(* Stoppen von Stationsfunktionen von rechter Arbeitsstation *)
	IF xStationStopWorkRight THEN
		(* Step  function station stop  *)
		CASE iStepAction OF
		(* Überprüfe zuerst welche Stationen gestoppt werden müssen  *)
		1:	iCheckStationNr:=1;
			ptrActivStation_FunctionStop:=ADR(TStation_Work_St1);
			iStepAction:=10;
		10:	IF (iCheckStationNr = 1) THEN ptrActivStation_FunctionStop:=ADR(TStation_Work_St1);
			ELSE
				iStepAction:=30;
				iCheckStationNr:=1;
				iStationNrReady:=0;
				RETURN;
			END_IF;
			xTmp:=	NOT(ptrActivStation_FunctionStop^.TControl.xDone)
					AND ptrActivStation_FunctionStop^.TControl.xRdy
					AND NOT(ptrActivStation_FunctionStop^.TControl.xExecute)
					AND NOT(ptrActivStation_FunctionStop^.TControl.xError)
					AND NOT(ptrActivStation_FunctionStop^.TControl.xStop);
			IF xTmp THEN
				(* Mindestens eine Station kann gestoppt werden *)
				iStepAction:=20;
			ELSE
				iCheckStationNr:=iCheckStationNr + 1;
			END_IF
		20:	ptrActivStation_FunctionStop^.TControl.xStop:=TRUE;
			iCheckStationNr:=iCheckStationNr + 1;
			(* next step *)
			iStepAction:=10;
		30:	IF (iCheckStationNr = 1) THEN ptrActivStation_FunctionStop:=ADR(TStation_Work_St1);END_IF;
			xTmp:=	(ptrActivStation_FunctionStop^.TControl.xDone OR ptrActivStation_FunctionStop^.TControl.xError)
					AND ptrActivStation_FunctionStop^.TControl.xRdy
					AND NOT(ptrActivStation_FunctionStop^.TControl.xExecute);
			IF xTmp THEN
				iStationNrReady:=iStationNrReady + 1;
			END_IF;
			iCheckStationNr:=iCheckStationNr + 1;
			IF (iCheckStationNr > 7) THEN
				IF (iStationNrReady = 7) THEN
					(* Alle Stationen sind gestoppt *)
					(* next step *)
					iStepAction:=40;
				ELSE
					(* Mindestens eine Station ist noch nicht gestoppt *)
					iCheckStationNr:=1;
					iStationNrReady:=0;
				END_IF;
			END_IF;
		(* Alle Stationen sind gestoppt. Nun müssen noch alle Achsen überprüft werden ob sie gestoppt sind *)
		40:	IF NOT(ptrTAxisZ_St1^.T_CtrleSingle.xNotMoving) AND NOT(ptrTAxisZ_St1^.T_CtrleSingle.xErr) THEN
				ptrTAxisZ_St1^.T_CtrleSingle.iFunction:=5;
				ptrTAxisZ_St1^.T_CtrleSingle.xExecute:=TRUE;
			END_IF;
			IF NOT(ptrTAxisS_St1^.T_CtrleSingle.xNotMoving) AND NOT(ptrTAxisS_St1^.T_CtrleSingle.xErr) THEN
				ptrTAxisS_St1^.T_CtrleSingle.iFunction:=5;
				ptrTAxisS_St1^.T_CtrleSingle.xExecute:=TRUE;
			END_IF;
			iStepAction:=50;
		(* Warte bis alle Achsen stehen *)
		50:	xTmp:=	(NOT(ptrTAxisZ_St1^.T_CtrleSingle.xExecute) AND (ptrTAxisZ_St1^.T_CtrleSingle.xDone OR ptrTAxisZ_St1^.T_CtrleSingle.xErr)) AND
					(NOT(ptrTAxisS_St1^.T_CtrleSingle.xExecute) AND (ptrTAxisS_St1^.T_CtrleSingle.xDone OR ptrTAxisS_St1^.T_CtrleSingle.xErr));
			IF xTmp THEN
				(* action done *)
				iStepAction:=90;
				T_ExchgParam.T_Visu.T_Message.iState:=274;	(* Warnung: Funktion wurde gestoppt ! *)
			END_IF;
		(* action done *)
		90:	T_Visu.T_CtrleAction.xFunctionActive:=FALSE;
			T_StartUp.T_State.xBlockChangeMovementVisu:=FALSE;
			T_Visu.T_CtrleAction.xDone:=TRUE;
			T_Visu.T_CtrleAction.xNotReady:=FALSE;
			T_Visu.T_CtrleAction.xErr:=FALSE;
			T_Visu.T_CtrleAction.udiErrorID:=0;
			xStationStopWorkRight:=FALSE;
		(* function not ready *)
		95:	T_StartUp.T_State.xBlockChangeMovementVisu:=FALSE;
			TimerNotReady(IN:=TRUE);
			xStationStopWorkRight:=FALSE;
		END_CASE;
	END_IF;
END_ACTION
ACTION VisuFunction_ToolCalibration:
(* Ausführen der Stationsfunktion für das Kalibrieren des ToolDefelction und ToolTorque *)
	IF xStationToolCalibrateFunction THEN
		(* Step  function station  *)
		CASE iStepAction OF
		(* Überprüfe zuerst ob es sich um die Station MicroHead oder Entgratstation handelt  *)
		1:	IF (T_ExchgParam.T_StationCommon.T_Param_StationWork.T_Fct_SpindleCalibration.iSelectCalibrationCylinder = 1) THEN
				ptrActivStation^.THWWorkStation.TCtrlWork.xActiveCalibrateToolDeflection:=TRUE;
				ptrActivStation^.THWWorkStation.TCtrlWork.xActiveCalibrateToolTorque:=FALSE;
			END_IF;
			IF (T_ExchgParam.T_StationCommon.T_Param_StationWork.T_Fct_SpindleCalibration.iSelectCalibrationCylinder = 2) THEN
				ptrActivStation^.THWWorkStation.TCtrlWork.xActiveCalibrateToolDeflection:=FALSE;
				ptrActivStation^.THWWorkStation.TCtrlWork.xActiveCalibrateToolTorque:=TRUE;
			END_IF;
			iStepAction:=10;
		(* check station state *)
		10:	xTmp:=	ptrActivStation^.TControl.xDone
					AND ptrActivStation^.TControl.xRdy
					AND NOT(ptrActivStation^.TControl.xExecute)
					AND NOT(ptrActivStation^.TControl.xError)
					AND NOT(ptrActivStation^.TControl.xStop);
			(* next step *)
			IF xTmp THEN iStepAction:=20; ELSE iStepAction:=95; END_IF
		(* determin function number *)
		20:	T_ExchgParam.T_Visu.T_Message.iState:=66;	(* Info: Kalibrierungsfunktion gestartet ! *)
			ptrActivStation^.TControl.iFunctNr:=7;
			ptrActivStation^.TControl.xExecute:=TRUE;
			ptrActivStation^.THWWorkStation.TCtrlWork.xStopToolRotation:=TRUE;
			iStepAction:=30;
			(* next step *)
			xStepActionDone:=FALSE;
		(* wait confirmation *)
		30:	IF NOT(xStepActionDone) THEN
			(* release execution *)
				ptrActivStation^.TControl.xExecute:=FALSE;
				xStepActionDone:=TRUE;
			ELSE
				T_ExchgParam.T_StationCommon.T_Param_StationWork.T_Fct_SpindleCalibration:=T_NovRAM.T_Parameter.T_StationWork[gciStationSt1].T_Fct_SpindleCalibration;
				IF (T_ExchgParam.T_StationCommon.T_Param_StationWork.T_Fct_SpindleCalibration.iSelectCalibrationCylinder = 1) THEN
					T_ExchgParam.T_StationCommon.T_Param_StationWork.T_Fct_SpindleCalibration.arOffsetToolDeflection[1]:=ptrActivStation^.THWWorkStation.TCtrlWork.rOffsetToolDeflection;
				END_IF;
				IF (T_ExchgParam.T_StationCommon.T_Param_StationWork.T_Fct_SpindleCalibration.iSelectCalibrationCylinder = 2) THEN
					T_ExchgParam.T_StationCommon.T_Param_StationWork.T_Fct_SpindleCalibration.arOffseTToolTorque[1]:=ptrActivStation^.THWWorkStation.TCtrlWork.rOffseTToolTorque;
				END_IF;
				IF ptrActivStation^.TControl.xDone THEN
					(* action done *)
					iStepAction:=40;
					xStepActionDone:=FALSE;
				END_IF
			END_IF
		40:	T_ExchgParam.T_StationCommon.T_Param_StationWork.T_Fct_SpindleCalibration:=T_NovRAM.T_Parameter.T_StationWork[gciStationSt1].T_Fct_SpindleCalibration;
			iStepAction:=50;
		50:	xAction_SaveNovRAM:=TRUE;
			xBlockSetNovRamAction_End:=TRUE;
			iStepActionNovRam:=1;
			iStepAction:=60;
		60:	IF NOT(xAction_SaveNovRAM) THEN
				T_ExchgParam.T_Visu.T_Message.iState:=67;	(* Info: Kalibrierungsfunktion beendet ! *)
				xUpdateStationParameter:=TRUE;
				iStepAction:=90;
			END_IF;
		(* action done *)
		90:	T_Visu.T_CtrleAction.xDone:=TRUE;
			T_Visu.T_CtrleAction.xNotReady:=FALSE;
			T_Visu.T_CtrleAction.xErr:=FALSE;
			T_Visu.T_CtrleAction.udiErrorID:=0;
			xStationToolCalibrateFunction:=FALSE;
		(* function not ready *)
		95:	TimerNotReady(IN:=TRUE);
			xStationToolCalibrateFunction:=FALSE;
		END_CASE
	END_IF

(* Spindelkalibrierung EIN/AUS *)
	IF xSpindelCalibrationONOFF THEN
		CASE iStepAction OF
		(* check state *)
		1:	xTmp:=	TRUE;
			(* next step *)
			IF xTmp THEN iStepAction:=10; ELSE iStepAction:=95; END_IF
		(* Set Value *)
		10:	gxSpindelCalibrationONOFF_St1:=NOT(gxSpindelCalibrationONOFF_St1);
			iStepAction:=90;
		(* action done *)
		90:	T_Visu.T_CtrleAction.xDone:=TRUE;
			T_Visu.T_CtrleAction.xNotReady:=FALSE;
			T_Visu.T_CtrleAction.xErr:=FALSE;
			T_Visu.T_CtrleAction.udiErrorID:=0;
			xSpindelCalibrationONOFF:=FALSE;
		(* cylinder not ready *)
		95:	TimerNotReady(IN:=TRUE);
			xSpindelCalibrationONOFF:=FALSE;
		END_CASE
	END_IF;

	IF (T_Visu.T_PlcParam.dwActualPage = gT_PageNumber.iWorkStation_Setup1) THEN
		IF (T_NovRAM.T_Parameter.T_StationWork[gciStationSt1].T_Fct_SpindleCalibration.iSelectCalibrationCylinder <> 1) AND
			(T_NovRAM.T_Parameter.T_StationWork[gciStationSt1].T_Fct_SpindleCalibration.iSelectCalibrationCylinder <> 2) THEN
			T_NovRAM.T_Parameter.T_StationWork[gciStationSt1].T_Fct_SpindleCalibration.iSelectCalibrationCylinder:=1;
		END_IF;
		IF (T_ExchgParam.T_StationCommon.T_Param_StationWork.T_Fct_SpindleCalibration.iSelectCalibrationCylinder <> 1) AND
			(T_ExchgParam.T_StationCommon.T_Param_StationWork.T_Fct_SpindleCalibration.iSelectCalibrationCylinder <> 2) THEN
			T_ExchgParam.T_StationCommon.T_Param_StationWork.T_Fct_SpindleCalibration.iSelectCalibrationCylinder:=1;
		END_IF;
		IF (T_ExchgParam.T_StationCommon.T_Param_StationWork.T_Fct_SpindleCalibration.iSelectCalibrationCylinder <>
		     T_NovRAM.T_Parameter.T_StationWork[gciStationSt1].T_Fct_SpindleCalibration.iSelectCalibrationCylinder) THEN
			T_NovRAM.T_Parameter.T_StationWork[gciStationSt1].T_Fct_SpindleCalibration.iSelectCalibrationCylinder:=
											T_ExchgParam.T_StationCommon.T_Param_StationWork.T_Fct_SpindleCalibration.iSelectCalibrationCylinder;
		END_IF;

		T_ExchgParam.T_StationCommon.T_Param_StationWork.T_Fct_SpindleCalibration.rEffectiveForceToolDeflection:=
					T_NovRAM.T_Parameter.T_StationWork[gciStationSt1].T_OnlineChange.rForceDeflection +
					T_NovRAM.T_Parameter.T_StationWork[gciStationSt1].T_Fct_SpindleCalibration.arOffsetToolDeflection[1];
		T_ExchgParam.T_StationCommon.T_Param_StationWork.T_Fct_SpindleCalibration.rNullValueToolDeflection:=
					T_NovRAM.T_Parameter.T_StationWork[gciStationSt1].T_OnlineChange.rForceDeflection;

		T_ExchgParam.T_StationCommon.T_Param_StationWork.T_Fct_SpindleCalibration.rEffectiveForceToolTorque:=
					T_NovRAM.T_Parameter.T_StationWork[gciStationSt1].T_OnlineChange.rTorqueLevelHC +
					T_NovRAM.T_Parameter.T_StationWork[gciStationSt1].T_Fct_SpindleCalibration.arOffseTToolTorque[1];
		T_ExchgParam.T_StationCommon.T_Param_StationWork.T_Fct_SpindleCalibration.rNullValueToolTorque:=
					T_NovRAM.T_Parameter.T_StationWork[gciStationSt1].T_OnlineChange.rTorqueLevelHC;

		IF NOT(xStationToolCalibrateFunction) THEN
			T_ExchgParam.T_StationCommon.T_Param_StationWork.T_Fct_SpindleCalibration.arOffsetToolDeflection:=
					T_NovRAM.T_Parameter.T_StationWork[gciStationSt1].T_Fct_SpindleCalibration.arOffsetToolDeflection;
			T_ExchgParam.T_StationCommon.T_Param_StationWork.T_Fct_SpindleCalibration.arOffseTToolTorque:=
					T_NovRAM.T_Parameter.T_StationWork[gciStationSt1].T_Fct_SpindleCalibration.arOffseTToolTorque;
		END_IF;
	END_IF;
END_ACTION
ACTION VisuFunction_ToolChange:
(* Resetten des Werkzeugwechsel für den Automatik für Station 1,2,3 und 4-->braucht mindestens den OperatorLevel oder für das setzen der berechneten Z EndPosition *)
	IF xProcessStation1ResetToolChange OR xZSaveEndPosCalc THEN
		CASE iStepAction OF
		(* Überprüfe zuerst ob mindestens der OperatorLevel gesetzt ist *)
		1:	IF (T_ExchgParam.T_Visu.T_Level.iActLevel < 1) THEN
				T_ExchgParam.T_Visu.T_Message.iState:=217;	(* Warnung: Mindestens OperatorLevel wird benötigt ! *)
				iStepAction:=90;
			ELSE
				iStepAction:=10;
			END_IF;
		10:	T_ExchgParam.T_Visu.T_Message.iState:=103;	(* Aufforderung: Speichern bestätigen <Enter>, abbrechen <Esc> ? *)
			iStepAction:=20;
		(* waiting for key <Enter> or <Esc> *)
		20:	IF RisingEdgeKeyPanel_Enter.Q THEN
				iStepAction:=30;
			ELSE
				IF RisingEdgeKeyPanel_Esc.Q THEN
					iStepAction:=90;
					T_ExchgParam.T_Visu.T_Message.iState:=202;	(* Warnung: Aktion abgebrochen ! *)
				END_IF
			END_IF
			(* An other message has been displayed *)
			IF (T_ExchgParam.T_Visu.T_Message.iState<>103) AND (T_ExchgParam.T_Visu.T_Message.iState<>202) THEN iStepAction:=90; END_IF
		30:	IF xProcessStation1ResetToolChange THEN
				T_NovRam.T_Parameter.T_StationWork[1].T_ToolCounter.diToolCycleCounter:=0;
				T_ExchgParam.T_StationCommon.T_ToolCounter_St1.diToolCycleCounter:=0;
				IF NOT(gxProcessCylindricalAreaActive) THEN
					garPositionEndProcCalc[1]:=T_NovRam.T_Parameter.T_StationWork[1].T_StProcess.rPositionEndProc;
					T_ExchgParam.T_StationCommon.rPositionEndProcCalc:=T_NovRam.T_Parameter.T_StationWork[1].T_StProcess.rPositionEndProc;
				ELSE
					garPositionEndProcCalc[1]:=T_NovRam.T_Parameter.T_StationWork[1].T_StProcess.rZPositionCylindricalArea;
					T_ExchgParam.T_StationCommon.rPositionEndProcCalc:=T_NovRam.T_Parameter.T_StationWork[1].T_StProcess.rZPositionCylindricalArea;
				END_IF;
				garCentringEndProcCalc[1]:=T_NovRam.T_Parameter.T_StationWork[1].T_StProcess.rCentringPosZ1Axis;
				T_ExchgParam.T_StationCommon.rCentringEndProcCalc:=T_NovRam.T_Parameter.T_StationWork[1].T_StProcess.rCentringPosZ1Axis;
			ELSE
				IF (T_ExchgParam.T_StationCommon.bSelectShowIncValue = 0) THEN
					garPositionEndProcCalc[1]:=T_ExchgParam.T_StationCommon.rPositionEndProcCalc;
				ELSE
					garCentringEndProcCalc[1]:=T_ExchgParam.T_StationCommon.rCentringEndProcCalc;
				END_IF;
			END_IF;
			iStepAction:=40;
		40:	IF xZSaveEndPosCalc THEN
				IF (T_ExchgParam.T_StationCommon.bSelectShowIncValue = 0) THEN
					IF (garPositionEndProcCalc[1] <> T_ExchgParam.T_StationCommon.rPositionEndProcCalc) THEN
						T_ExchgParam.T_StationCommon.rPositionEndProcCalc:=garPositionEndProcCalc[1];
					END_IF;
				ELSE
					IF (garCentringEndProcCalc[1] <> T_ExchgParam.T_StationCommon.rCentringEndProcCalc) THEN
						T_ExchgParam.T_StationCommon.rCentringEndProcCalc:=garCentringEndProcCalc[1];
					END_IF;
				END_IF;
			END_IF;
			xAction_SaveNovRAM:=TRUE;
			xBlockSetNovRamAction_End:=TRUE;
			iStepActionNovRam:=1;
			iStepAction:=50;
		50:	IF NOT(xAction_SaveNovRAM) THEN
				iStepAction:=90;
				IF xProcessStation1ResetToolChange THEN
					T_ExchgParam.T_Visu.T_Message.iState:=68;	(* Info: WzZähler für Station 1 wurde zurückgesetzt ! *)
				ELSE
					T_ExchgParam.T_Visu.T_Message.iState:=69;	(* Info: Position gespeichert ! *)
				END_IF;
			END_IF;
		(* axis not ready *)
		95:	TimerNotReady(IN:=TRUE);
			xProcessStation1ResetToolChange:=xZSaveEndPosCalc:=FALSE;
		(* slow/fast configuration done *)
		90:	T_Visu.T_CtrleAction.xDone:=TRUE;
			T_Visu.T_CtrleAction.xNotReady:=FALSE;
			T_Visu.T_CtrleAction.xErr:=FALSE;
			T_Visu.T_CtrleAction.udiErrorID:=0;
			xProcessStation1ResetToolChange:=xZSaveEndPosCalc:=FALSE;
		END_CASE
	END_IF;


(* Umschalten Z Ink Wert für Bearbeitung oder Zentrierung *)
	IF xSelectZInkWorkInfo OR xSelectZInkCentringInfo THEN
		CASE iStepAction OF
		(* Überprüfe zuerst ob mindestens der OperatorLevel gesetzt ist *)
		1:	iStepAction:=10;
		10:	IF xSelectZInkWorkInfo THEN
				T_ExchgParam.T_StationCommon.bSelectShowIncValue:=0;
			ELSE
				T_ExchgParam.T_StationCommon.bSelectShowIncValue:=1;
			END_IF;
			iStepAction:=90;
		(* axis not ready *)
		95:	TimerNotReady(IN:=TRUE);
			xSelectZInkWorkInfo:=xSelectZInkCentringInfo:=FALSE;
		(* slow/fast configuration done *)
		90:	T_Visu.T_CtrleAction.xDone:=TRUE;
			T_Visu.T_CtrleAction.xNotReady:=FALSE;
			T_Visu.T_CtrleAction.xErr:=FALSE;
			T_Visu.T_CtrleAction.udiErrorID:=0;
			xSelectZInkWorkInfo:=xSelectZInkCentringInfo:=FALSE;
		END_CASE
	END_IF;
END_ACTION
ACTION VisuUpdateParameter:
IF (T_Visu.T_PlcParam.dwActualPage = gT_PageNumber.iHandMode_OnlineChange) THEN
	xFctUpdateOnlineChangeValue(	ptrProfileOnlineChange:=ADR(T_Profile.T_Profile_MinMax),
									ptrProfileOnlineChangeLoad:=ADR(T_Profile.T_LoadProfileParameter.T_ProfileOnlineChange),
									ptrExchgParamStationCommon:=ADR(T_ExchgParam.T_ProfileCommon.T_OnlineChange),
									TOnlineChangeParameter:=T_NovRam.T_Parameter.T_StationWork[gciStationSt1].T_OnlineChange);
END_IF;
END_ACTION

(* POU PRG_LAYER5_VISU/FB_VISU/FBQVIS_INITPAGE, ST *)
FUNCTION_BLOCK FBQVIS_INITPAGE
VAR_INPUT
END_VAR
VAR_OUTPUT
END_VAR
VAR_IN_OUT
	T_Visu:ST_QVIS;
END_VAR
VAR
(* pointer *)
	ptrConfigPage: POINTER TO ST_CONFIGPAGE;
(* variable *)
	iIndexPage:INT;
	iPageNumber:INT;
(* variable Tmp *)
	i:INT;
END_VAR
(****************************************************************************************************************************************************)
(***********                    This Functionblock init all the defined page in QVis for the hole page management                            ************)
(****************************************************************************************************************************************************)
(* init. index array *)
FOR i:=0 TO 999 DO
	T_Visu.T_PageIndex[i].iIndexConfigPage:=0;
END_FOR

(* init. Number Page *)
iPageNumber:=0;
Page_000_Start;
Page_001_BIOS;
Page_002_BIOS;
Page_010_AutoMode_Process;
Page_011_AutoMode_ProcessValue1;
Page_012_AutoMode_ProcessValue2;	(* IGS *)
Page_013_AutoMode_PartQuality;
Page_020_AutoMode_Referencing;
Page_030_AutoMode_Profile;
Page_040_AutoMode_ToolChange;
Page_041_AutoMode_UserLevel;
Page_042_AutoMode_Language;
Page_050_AutoMode_WPCounter;
Page_051_AutoMode_LampTest;
Page_052_AutoMode_SafetyCheck;
Page_053_AutoMode_SysInfo;
Page_060_AutoMode_ErrorList;
Page_070_AutoMode_Parameter;
Page_110_HandMode_Process;
Page_111_HandMode_WorkParameter;		(* IGS *)
Page_112_HandMode_RegulatorPara;		(* IGS *)
Page_113_HandMode_OnlineChange;
Page_114_HandMode_ConfigPosition;
Page_120_HandMode_ProfileMngmt1;
Page_150_HandMode_Setup1;
Page_160_HandMode_ErrorList;
Page_170_HandMode_Parameter;
Page_210_WorkStation_Axis1;
Page_220_WorkStation_Cylinder1;
Page_230_WorkStation_Valve1;
Page_240_WorkStation_Function1;
Page_250_WorkStation_Setup1;
Page_251_WorkStation_Setup2;
Page_252_WorkStation_Setup3;
Page_253_WorkStation_Setup4;
Page_254_WorkStation_Setup5;
Page_260_WorkStation_ErrorList;
Page_270_WorkStation_Parameter;
END_FUNCTION_BLOCK
ACTION Page_000_Start:
(* QVis page 0, start page *)
iIndexPage:=gT_PageNumber.iStart_Page1;
iPageNumber:=iPageNumber+1;
T_Visu.T_PageIndex[iIndexPage].iIndexConfigPage:=iPageNumber;
ptrConfigPage:=ADR(T_Visu.T_ConfigPage[T_Visu.T_PageIndex[iIndexPage].iIndexConfigPage]);
ptrConfigPage^.sName:='Start page';
ptrConfigPage^.wMaskBtPanelLeft:=16#0;
ptrConfigPage^.wMaskBtPanelRight:=16#0;
ptrConfigPage^.wMaskFunctionPanel:=16#0;
(* Navigation panel restriction *)
ptrConfigPage^.wMaskTouchScreenNavPanel:=16#0;
(* Process mask *)
ptrConfigPage^.wMaskProcBtPanelLeft:=16#0;
ptrConfigPage^.wMaskProcBtPanelRight:=16#0;
ptrConfigPage^.wMaskProcFunctionPanel:=16#0;
(* Button edge action *)
ptrConfigPage^.aiRTrigActionPanelLeft[1]:=0;
ptrConfigPage^.aiRTrigActionPanelLeft[2]:=0;
ptrConfigPage^.aiRTrigActionPanelLeft[3]:=0;
ptrConfigPage^.aiRTrigActionPanelLeft[4]:=0;
ptrConfigPage^.aiRTrigActionPanelLeft[5]:=0;
ptrConfigPage^.aiRTrigActionPanelRight[1]:=0;
ptrConfigPage^.aiRTrigActionPanelRight[2]:=0;
ptrConfigPage^.aiRTrigActionPanelRight[3]:=0;
ptrConfigPage^.aiRTrigActionPanelRight[4]:=0;
ptrConfigPage^.aiRTrigActionPanelRight[5]:=0;
ptrConfigPage^.aiFTrigActionPanelRight[1]:=0;
ptrConfigPage^.aiFTrigActionPanelRight[2]:=0;
ptrConfigPage^.aiFTrigActionPanelRight[3]:=0;
ptrConfigPage^.aiFTrigActionPanelRight[4]:=0;
ptrConfigPage^.aiFTrigActionPanelRight[5]:=0;
ptrConfigPage^.aiRTrigActionFunctionPanel[1]:=0;
ptrConfigPage^.aiRTrigActionFunctionPanel[2]:=0;
ptrConfigPage^.aiRTrigActionFunctionPanel[3]:=0;
ptrConfigPage^.aiRTrigActionFunctionPanel[4]:=0;
ptrConfigPage^.aiRTrigActionFunctionPanel[5]:=0;
ptrConfigPage^.aiRTrigActionFunctionPanel[6]:=0;
ptrConfigPage^.aiRTrigActionFunctionPanel[7]:=0;
ptrConfigPage^.aiRTrigActionFunctionPanel[8]:=0;
ptrConfigPage^.aiRTrigActionFunctionPanel[9]:=0;
ptrConfigPage^.aiRTrigActionFunctionPanel[10]:=0;
ptrConfigPage^.aiRTrigActionFunctionPanel[11]:=0;
ptrConfigPage^.aiRTrigActionFunctionPanel[12]:=0;
ptrConfigPage^.aiRTrigActionTouchScreenNavPanel[1,1]:=0;
ptrConfigPage^.aiRTrigActionTouchScreenNavPanel[1,2]:=0;
ptrConfigPage^.aiRTrigActionTouchScreenNavPanel[1,3]:=0;
ptrConfigPage^.aiRTrigActionTouchScreenNavPanel[1,4]:=0;
ptrConfigPage^.aiRTrigActionTouchScreenNavPanel[1,5]:=0;
ptrConfigPage^.aiRTrigActionTouchScreenNavPanel[1,6]:=0;
ptrConfigPage^.aiRTrigActionTouchScreenNavPanel[1,7]:=0;
ptrConfigPage^.aiRTrigActionTouchScreenNavPanel[1,8]:=0;
ptrConfigPage^.aiRTrigActionTouchScreenNavPanel[1,9]:=0;
ptrConfigPage^.aiRTrigActionTouchScreenNavPanel[2,1]:=0;
ptrConfigPage^.aiRTrigActionTouchScreenNavPanel[2,2]:=0;
ptrConfigPage^.aiRTrigActionTouchScreenNavPanel[2,3]:=0;
ptrConfigPage^.aiRTrigActionTouchScreenNavPanel[2,4]:=0;
ptrConfigPage^.aiRTrigActionTouchScreenNavPanel[2,5]:=0;
ptrConfigPage^.aiRTrigActionTouchScreenNavPanel[2,6]:=0;
ptrConfigPage^.aiRTrigActionTouchScreenNavPanel[2,7]:=0;
ptrConfigPage^.aiRTrigActionTouchScreenNavPanel[2,8]:=0;
ptrConfigPage^.aiRTrigActionTouchScreenNavPanel[2,9]:=0;
ptrConfigPage^.aiRTrigActionTouchScreenNavPanel[3,1]:=0;
ptrConfigPage^.aiRTrigActionTouchScreenNavPanel[3,2]:=0;
ptrConfigPage^.aiRTrigActionTouchScreenNavPanel[3,3]:=0;
ptrConfigPage^.aiRTrigActionTouchScreenNavPanel[3,4]:=0;
ptrConfigPage^.aiRTrigActionTouchScreenNavPanel[3,5]:=0;
ptrConfigPage^.aiRTrigActionTouchScreenNavPanel[3,6]:=0;
ptrConfigPage^.aiRTrigActionTouchScreenNavPanel[3,7]:=0;
ptrConfigPage^.aiRTrigActionTouchScreenNavPanel[3,8]:=0;
ptrConfigPage^.aiRTrigActionTouchScreenNavPanel[3,9]:=0;
ptrConfigPage^.aiRTrigActionTouchScreenNavPanel[4,1]:=0;
ptrConfigPage^.aiRTrigActionTouchScreenNavPanel[4,2]:=0;
ptrConfigPage^.aiRTrigActionTouchScreenNavPanel[4,3]:=0;
ptrConfigPage^.aiRTrigActionTouchScreenNavPanel[4,4]:=0;
ptrConfigPage^.aiRTrigActionTouchScreenNavPanel[4,5]:=0;
ptrConfigPage^.aiRTrigActionTouchScreenNavPanel[4,6]:=0;
ptrConfigPage^.aiRTrigActionTouchScreenNavPanel[4,7]:=0;
ptrConfigPage^.aiRTrigActionTouchScreenNavPanel[4,8]:=0;
ptrConfigPage^.aiRTrigActionTouchScreenNavPanel[4,9]:=0;
ptrConfigPage^.aiRTrigActionTouchScreenNavPanel[5,1]:=0;
ptrConfigPage^.aiRTrigActionTouchScreenNavPanel[5,2]:=0;
ptrConfigPage^.aiRTrigActionTouchScreenNavPanel[5,3]:=0;
ptrConfigPage^.aiRTrigActionTouchScreenNavPanel[5,4]:=0;
ptrConfigPage^.aiRTrigActionTouchScreenNavPanel[5,5]:=0;
ptrConfigPage^.aiRTrigActionTouchScreenNavPanel[5,6]:=0;
ptrConfigPage^.aiRTrigActionTouchScreenNavPanel[5,7]:=0;
ptrConfigPage^.aiRTrigActionTouchScreenNavPanel[5,8]:=0;
ptrConfigPage^.aiRTrigActionTouchScreenNavPanel[5,9]:=0;
ptrConfigPage^.aiRTrigActionTouchScreenNavPanel[6,1]:=0;
ptrConfigPage^.aiRTrigActionTouchScreenNavPanel[6,2]:=0;
ptrConfigPage^.aiRTrigActionTouchScreenNavPanel[6,3]:=0;
ptrConfigPage^.aiRTrigActionTouchScreenNavPanel[6,4]:=0;
ptrConfigPage^.aiRTrigActionTouchScreenNavPanel[6,5]:=0;
ptrConfigPage^.aiRTrigActionTouchScreenNavPanel[6,6]:=0;
ptrConfigPage^.aiRTrigActionTouchScreenNavPanel[6,7]:=0;
ptrConfigPage^.aiRTrigActionTouchScreenNavPanel[6,8]:=0;
ptrConfigPage^.aiRTrigActionTouchScreenNavPanel[6,9]:=0;
ptrConfigPage^.xMaskBtStart:=TRUE;
ptrConfigPage^.xMaskBtStop:=FALSE;
END_ACTION
ACTION Page_001_BIOS:
(* QVis page 1, BIOS input Password *)
iIndexPage:=gT_PageNumber.iBIOS_Page1;
iPageNumber:=iPageNumber+1;
T_Visu.T_PageIndex[iIndexPage].iIndexConfigPage:=iPageNumber;
ptrConfigPage:=ADR(T_Visu.T_ConfigPage[T_Visu.T_PageIndex[iIndexPage].iIndexConfigPage]);
ptrConfigPage^.sName:='BIOS input Password';
ptrConfigPage^.wMaskBtPanelLeft:=16#0;
ptrConfigPage^.wMaskBtPanelRight:=16#0;
ptrConfigPage^.wMaskFunctionPanel:=16#0;
(* Navigation panel restriction *)
ptrConfigPage^.wMaskTouchScreenNavPanel:=16#0;
(* Process mask *)
ptrConfigPage^.wMaskProcBtPanelLeft:=16#0;
ptrConfigPage^.wMaskProcBtPanelRight:=16#0;
ptrConfigPage^.wMaskProcFunctionPanel:=16#0;
(* Button edge action *)
ptrConfigPage^.aiRTrigActionPanelLeft[1]:=0;
ptrConfigPage^.aiRTrigActionPanelLeft[2]:=0;
ptrConfigPage^.aiRTrigActionPanelLeft[3]:=0;
ptrConfigPage^.aiRTrigActionPanelLeft[4]:=0;
ptrConfigPage^.aiRTrigActionPanelLeft[5]:=0;
ptrConfigPage^.aiRTrigActionPanelRight[1]:=0;
ptrConfigPage^.aiRTrigActionPanelRight[2]:=0;
ptrConfigPage^.aiRTrigActionPanelRight[3]:=0;
ptrConfigPage^.aiRTrigActionPanelRight[4]:=0;
ptrConfigPage^.aiRTrigActionPanelRight[5]:=0;
ptrConfigPage^.aiFTrigActionPanelRight[1]:=0;
ptrConfigPage^.aiFTrigActionPanelRight[2]:=0;
ptrConfigPage^.aiFTrigActionPanelRight[3]:=0;
ptrConfigPage^.aiFTrigActionPanelRight[4]:=0;
ptrConfigPage^.aiFTrigActionPanelRight[5]:=0;
ptrConfigPage^.aiRTrigActionFunctionPanel[1]:=0;
ptrConfigPage^.aiRTrigActionFunctionPanel[2]:=0;
ptrConfigPage^.aiRTrigActionFunctionPanel[3]:=0;
ptrConfigPage^.aiRTrigActionFunctionPanel[4]:=0;
ptrConfigPage^.aiRTrigActionFunctionPanel[5]:=0;
ptrConfigPage^.aiRTrigActionFunctionPanel[6]:=0;
ptrConfigPage^.aiRTrigActionFunctionPanel[7]:=0;
ptrConfigPage^.aiRTrigActionFunctionPanel[8]:=0;
ptrConfigPage^.aiRTrigActionFunctionPanel[9]:=0;
ptrConfigPage^.aiRTrigActionFunctionPanel[10]:=0;
ptrConfigPage^.aiRTrigActionFunctionPanel[11]:=0;
ptrConfigPage^.aiRTrigActionFunctionPanel[12]:=0;
TaskBar_BIOS;
ptrConfigPage^.xMaskBtStart:=FALSE;
ptrConfigPage^.xMaskBtStop:=FALSE;
END_ACTION
ACTION Page_002_BIOS:
(* QVis page 2, BIOS Parameter *)
iIndexPage:=gT_PageNumber.iBIOS_Page2;
iPageNumber:=iPageNumber+1;
T_Visu.T_PageIndex[iIndexPage].iIndexConfigPage:=iPageNumber;
ptrConfigPage:=ADR(T_Visu.T_ConfigPage[T_Visu.T_PageIndex[iIndexPage].iIndexConfigPage]);
ptrConfigPage^.sName:='BIOS Parameter';
ptrConfigPage^.wMaskBtPanelLeft:=16#0;
ptrConfigPage^.wMaskBtPanelRight:=16#0;
ptrConfigPage^.wMaskFunctionPanel:=16#0;
(* Navigation panel restriction *)
ptrConfigPage^.wMaskTouchScreenNavPanel:=16#0;
(* Process mask *)
ptrConfigPage^.wMaskProcBtPanelLeft:=16#0;
ptrConfigPage^.wMaskProcBtPanelRight:=16#0;
ptrConfigPage^.wMaskProcFunctionPanel:=16#0;
(* Button edge action *)
ptrConfigPage^.aiRTrigActionPanelLeft[1]:=0;
ptrConfigPage^.aiRTrigActionPanelLeft[2]:=0;
ptrConfigPage^.aiRTrigActionPanelLeft[3]:=0;
ptrConfigPage^.aiRTrigActionPanelLeft[4]:=0;
ptrConfigPage^.aiRTrigActionPanelLeft[5]:=0;
ptrConfigPage^.aiRTrigActionPanelRight[1]:=0;
ptrConfigPage^.aiRTrigActionPanelRight[2]:=0;
ptrConfigPage^.aiRTrigActionPanelRight[3]:=0;
ptrConfigPage^.aiRTrigActionPanelRight[4]:=0;
ptrConfigPage^.aiRTrigActionPanelRight[5]:=0;
ptrConfigPage^.aiFTrigActionPanelRight[1]:=0;
ptrConfigPage^.aiFTrigActionPanelRight[2]:=0;
ptrConfigPage^.aiFTrigActionPanelRight[3]:=0;
ptrConfigPage^.aiFTrigActionPanelRight[4]:=0;
ptrConfigPage^.aiFTrigActionPanelRight[5]:=0;
ptrConfigPage^.aiRTrigActionFunctionPanel[1]:=0;
ptrConfigPage^.aiRTrigActionFunctionPanel[2]:=0;
ptrConfigPage^.aiRTrigActionFunctionPanel[3]:=0;
ptrConfigPage^.aiRTrigActionFunctionPanel[4]:=0;
ptrConfigPage^.aiRTrigActionFunctionPanel[5]:=0;
ptrConfigPage^.aiRTrigActionFunctionPanel[6]:=0;
ptrConfigPage^.aiRTrigActionFunctionPanel[7]:=0;
ptrConfigPage^.aiRTrigActionFunctionPanel[8]:=0;
ptrConfigPage^.aiRTrigActionFunctionPanel[9]:=0;
ptrConfigPage^.aiRTrigActionFunctionPanel[10]:=0;
ptrConfigPage^.aiRTrigActionFunctionPanel[11]:=0;
ptrConfigPage^.aiRTrigActionFunctionPanel[12]:=0;
TaskBar_BIOS;
ptrConfigPage^.xMaskBtStart:=FALSE;
ptrConfigPage^.xMaskBtStop:=FALSE;
END_ACTION
ACTION Page_010_AutoMode_Process:
(* QVis page 10, AutoMode Process all holes *)
iIndexPage:=gT_PageNumber.iAutoMode_Process;
iPageNumber:=iPageNumber+1;
T_Visu.T_PageIndex[iIndexPage].iIndexConfigPage:=iPageNumber;
ptrConfigPage:=ADR(T_Visu.T_ConfigPage[T_Visu.T_PageIndex[iIndexPage].iIndexConfigPage]);
ptrConfigPage^.sName:='AutoMode Process all holes';
ptrConfigPage^.wMaskBtPanelLeft:=16#18;		(*              1 1000	Lampe & Parameter *)
ptrConfigPage^.wMaskBtPanelRight:=16#3E0;		(* 11 1110 0000	Auto Process, Work Info1, Work Info 2, WP Analysis, Meldung Anzeigen *)	(* alt: 1E0; *)
ptrConfigPage^.wMaskFunctionPanel:=16#1F;		(* F1, F2, F3, F4, F5 *)
(* Process mask *)
ptrConfigPage^.wMaskProcBtPanelLeft:=16#F;		(*              1 1111 *)
ptrConfigPage^.wMaskProcBtPanelRight:=16#3E0;	(* 11 1110 0000 Auto Process, Work Info1, Work Info 2, WP Analysis, Meldung Anzeigen *)	(* alt: 1E0; *)
ptrConfigPage^.wMaskProcFunctionPanel:=16#1;		(* F1 *)
(* Button edge action *)
ptrConfigPage^.aiRTrigActionPanelLeft[1]:=0;
ptrConfigPage^.aiRTrigActionPanelLeft[2]:=0;
ptrConfigPage^.aiRTrigActionPanelLeft[3]:=0;
ptrConfigPage^.aiRTrigActionPanelLeft[4]:=0;
ptrConfigPage^.aiRTrigActionPanelLeft[5]:=11000 + gT_PageNumber.iAutoMode_Parameter;		(* Parameter Page *)
ptrConfigPage^.aiRTrigActionPanelRight[1]:=10000 + gT_PageNumber.iAutoMode_Process;
ptrConfigPage^.aiRTrigActionPanelRight[2]:=10000 + gT_PageNumber.iAutoMode_ProcessValue1;
ptrConfigPage^.aiRTrigActionPanelRight[3]:=10000 + gT_PageNumber.iAutoMode_ProcessValue2;
ptrConfigPage^.aiRTrigActionPanelRight[4]:=10000 + gT_PageNumber.iAutoMode_PartQuality;
ptrConfigPage^.aiRTrigActionPanelRight[5]:=104;		(* Meldungsfenster Öffnen *)
ptrConfigPage^.aiFTrigActionPanelRight[1]:=0;
ptrConfigPage^.aiFTrigActionPanelRight[2]:=0;
ptrConfigPage^.aiFTrigActionPanelRight[3]:=0;
ptrConfigPage^.aiFTrigActionPanelRight[4]:=0;
ptrConfigPage^.aiFTrigActionPanelRight[5]:=0;
ptrConfigPage^.aiRTrigActionFunctionPanel[1]:=151;	(* Endlos Prozess für Messe *)
ptrConfigPage^.aiRTrigActionFunctionPanel[2]:=152;	(* Zentrieren EIN/AUS *)
ptrConfigPage^.aiRTrigActionFunctionPanel[3]:=153;	(* NurZentrieren EIN/AUS *)
ptrConfigPage^.aiRTrigActionFunctionPanel[4]:=154;	(* Suspension EIN/AUS *)
ptrConfigPage^.aiRTrigActionFunctionPanel[5]:=155;	(* WPUnfix EIN/AUS *)
ptrConfigPage^.aiRTrigActionFunctionPanel[6]:=0;
ptrConfigPage^.aiRTrigActionFunctionPanel[7]:=0;
ptrConfigPage^.aiRTrigActionFunctionPanel[8]:=0;
ptrConfigPage^.aiRTrigActionFunctionPanel[9]:=0;
ptrConfigPage^.aiRTrigActionFunctionPanel[10]:=0;
ptrConfigPage^.aiRTrigActionFunctionPanel[11]:=0;
ptrConfigPage^.aiRTrigActionFunctionPanel[12]:=0;
TaskBar_NormalMode;
ptrConfigPage^.xMaskBtStart:=TRUE;
ptrConfigPage^.xMaskBtStop:=TRUE;
END_ACTION
ACTION Page_011_AutoMode_ProcessValue1:
(* QVis page 11, AutoMode PartQuality *)
iIndexPage:=gT_PageNumber.iAutoMode_ProcessValue1;
iPageNumber:=iPageNumber+1;
T_Visu.T_PageIndex[iIndexPage].iIndexConfigPage:=iPageNumber;
ptrConfigPage:=ADR(T_Visu.T_ConfigPage[T_Visu.T_PageIndex[iIndexPage].iIndexConfigPage]);
ptrConfigPage^.sName:='AutoMode ProcessValue';
ptrConfigPage^.wMaskBtPanelLeft:=16#18;		(*              1 1000	Lampe & Parameter *)
ptrConfigPage^.wMaskBtPanelRight:=16#3E0;		(* 11 1110 0000	Auto Process, Work Info1, Work Info 2, WP Analysis, Meldung Anzeigen *)	(* alt: 1E0; *)
ptrConfigPage^.wMaskFunctionPanel:=16#0;
(* Process mask *)
ptrConfigPage^.wMaskProcBtPanelLeft:=16#F;		(*              1 1111 *)
ptrConfigPage^.wMaskProcBtPanelRight:=16#3E0;	(* 11 1110 0000 Auto Process, Work Info1, Work Info 2, WP Analysis, Meldung Anzeigen *)	(* alt: 1E0; *)
ptrConfigPage^.wMaskProcFunctionPanel:=16#0;
(* Button edge action *)
ptrConfigPage^.aiRTrigActionPanelLeft[1]:=0;
ptrConfigPage^.aiRTrigActionPanelLeft[2]:=0;
ptrConfigPage^.aiRTrigActionPanelLeft[3]:=0;
ptrConfigPage^.aiRTrigActionPanelLeft[4]:=0;
ptrConfigPage^.aiRTrigActionPanelLeft[5]:=11000 + gT_PageNumber.iAutoMode_Parameter;		(* Parameter Page *)
ptrConfigPage^.aiRTrigActionPanelRight[1]:=10000 + gT_PageNumber.iAutoMode_Process;
ptrConfigPage^.aiRTrigActionPanelRight[2]:=10000 + gT_PageNumber.iAutoMode_ProcessValue1;
ptrConfigPage^.aiRTrigActionPanelRight[3]:=10000 + gT_PageNumber.iAutoMode_ProcessValue2;
ptrConfigPage^.aiRTrigActionPanelRight[4]:=10000 + gT_PageNumber.iAutoMode_PartQuality;
ptrConfigPage^.aiRTrigActionPanelRight[5]:=104;		(* Meldungsfenster Öffnen *)
ptrConfigPage^.aiFTrigActionPanelRight[1]:=0;
ptrConfigPage^.aiFTrigActionPanelRight[2]:=0;
ptrConfigPage^.aiFTrigActionPanelRight[3]:=0;
ptrConfigPage^.aiFTrigActionPanelRight[4]:=0;
ptrConfigPage^.aiFTrigActionPanelRight[5]:=0;
ptrConfigPage^.aiRTrigActionFunctionPanel[1]:=0;
ptrConfigPage^.aiRTrigActionFunctionPanel[2]:=0;
ptrConfigPage^.aiRTrigActionFunctionPanel[3]:=0;
ptrConfigPage^.aiRTrigActionFunctionPanel[4]:=0;
ptrConfigPage^.aiRTrigActionFunctionPanel[5]:=0;
ptrConfigPage^.aiRTrigActionFunctionPanel[6]:=0;
ptrConfigPage^.aiRTrigActionFunctionPanel[7]:=0;
ptrConfigPage^.aiRTrigActionFunctionPanel[8]:=0;
ptrConfigPage^.aiRTrigActionFunctionPanel[9]:=0;
ptrConfigPage^.aiRTrigActionFunctionPanel[10]:=0;
ptrConfigPage^.aiRTrigActionFunctionPanel[11]:=0;
ptrConfigPage^.aiRTrigActionFunctionPanel[12]:=0;
TaskBar_NormalMode;
ptrConfigPage^.xMaskBtStart:=TRUE;
ptrConfigPage^.xMaskBtStop:=TRUE;
END_ACTION
ACTION Page_012_AutoMode_ProcessValue2:
(* QVis page 12, AutoMode ProzessValue2 *)
iIndexPage:=gT_PageNumber.iAutoMode_ProcessValue2;
iPageNumber:=iPageNumber+1;
T_Visu.T_PageIndex[iIndexPage].iIndexConfigPage:=iPageNumber;
ptrConfigPage:=ADR(T_Visu.T_ConfigPage[T_Visu.T_PageIndex[iIndexPage].iIndexConfigPage]);
ptrConfigPage^.sName:='AutoMode ProcessValue2';
ptrConfigPage^.wMaskBtPanelLeft:=16#18;		(*              1 1000	Lampe & Parameter *)
ptrConfigPage^.wMaskBtPanelRight:=16#3E0;		(* 11 1110 0000	Auto Process, Work Info1, Work Info 2, WP Analysis, Meldung Anzeigen *)	(* alt: 1E0; *)
ptrConfigPage^.wMaskFunctionPanel:=16#0;
(* Process mask *)
ptrConfigPage^.wMaskProcBtPanelLeft:=16#F;		(*              1 1111 *)
ptrConfigPage^.wMaskProcBtPanelRight:=16#3E0;	(* 11 1110 0000 Auto Process, Work Info1, Work Info 2, WP Analysis, Meldung Anzeigen *)	(* alt: 1E0; *)
ptrConfigPage^.wMaskProcFunctionPanel:=16#0;
(* Button edge action *)
ptrConfigPage^.aiRTrigActionPanelLeft[1]:=0;
ptrConfigPage^.aiRTrigActionPanelLeft[2]:=0;
ptrConfigPage^.aiRTrigActionPanelLeft[3]:=0;
ptrConfigPage^.aiRTrigActionPanelLeft[4]:=0;
ptrConfigPage^.aiRTrigActionPanelLeft[5]:=11000 + gT_PageNumber.iAutoMode_Parameter;		(* Parameter Page *)
ptrConfigPage^.aiRTrigActionPanelRight[1]:=10000 + gT_PageNumber.iAutoMode_Process;
ptrConfigPage^.aiRTrigActionPanelRight[2]:=10000 + gT_PageNumber.iAutoMode_ProcessValue1;
ptrConfigPage^.aiRTrigActionPanelRight[3]:=10000 + gT_PageNumber.iAutoMode_ProcessValue2;
ptrConfigPage^.aiRTrigActionPanelRight[4]:=10000 + gT_PageNumber.iAutoMode_PartQuality;
ptrConfigPage^.aiRTrigActionPanelRight[5]:=104;		(* Meldungsfenster Öffnen *)
ptrConfigPage^.aiFTrigActionPanelRight[1]:=0;
ptrConfigPage^.aiFTrigActionPanelRight[2]:=0;
ptrConfigPage^.aiFTrigActionPanelRight[3]:=0;
ptrConfigPage^.aiFTrigActionPanelRight[4]:=0;
ptrConfigPage^.aiFTrigActionPanelRight[5]:=0;
ptrConfigPage^.aiRTrigActionFunctionPanel[1]:=0;
ptrConfigPage^.aiRTrigActionFunctionPanel[2]:=0;
ptrConfigPage^.aiRTrigActionFunctionPanel[3]:=0;
ptrConfigPage^.aiRTrigActionFunctionPanel[4]:=0;
ptrConfigPage^.aiRTrigActionFunctionPanel[5]:=0;
ptrConfigPage^.aiRTrigActionFunctionPanel[6]:=0;
ptrConfigPage^.aiRTrigActionFunctionPanel[7]:=0;
ptrConfigPage^.aiRTrigActionFunctionPanel[8]:=0;
ptrConfigPage^.aiRTrigActionFunctionPanel[9]:=0;
ptrConfigPage^.aiRTrigActionFunctionPanel[10]:=0;
ptrConfigPage^.aiRTrigActionFunctionPanel[11]:=0;
ptrConfigPage^.aiRTrigActionFunctionPanel[12]:=0;
TaskBar_NormalMode;
ptrConfigPage^.xMaskBtStart:=TRUE;
ptrConfigPage^.xMaskBtStop:=TRUE;
END_ACTION
ACTION Page_013_AutoMode_PartQuality:
(* QVis page 12, AutoMode PartQuality *)
iIndexPage:=gT_PageNumber.iAutoMode_PartQuality;
iPageNumber:=iPageNumber+1;
T_Visu.T_PageIndex[iIndexPage].iIndexConfigPage:=iPageNumber;
ptrConfigPage:=ADR(T_Visu.T_ConfigPage[T_Visu.T_PageIndex[iIndexPage].iIndexConfigPage]);
ptrConfigPage^.sName:='AutoMode PartQuality';
ptrConfigPage^.wMaskBtPanelLeft:=16#18;		(*              1 1000	Lampe & Parameter *)
ptrConfigPage^.wMaskBtPanelRight:=16#3E0;		(* 11 1110 0000	Auto Process, Work Info1, Work Info 2, WP Analysis, Meldung Anzeigen *)	(* alt: 1E0; *)
ptrConfigPage^.wMaskFunctionPanel:=16#1;
(* Process mask *)
ptrConfigPage^.wMaskProcBtPanelLeft:=16#F;		(*              1 1111 *)
ptrConfigPage^.wMaskProcBtPanelRight:=16#3E0;	(* 11 1110 0000 Auto Process, Work Info1, Work Info 2, WP Analysis, Meldung Anzeigen *)	(* alt: 1E0; *)
ptrConfigPage^.wMaskProcFunctionPanel:=16#0;
(* Button edge action *)
ptrConfigPage^.aiRTrigActionPanelLeft[1]:=0;
ptrConfigPage^.aiRTrigActionPanelLeft[2]:=0;
ptrConfigPage^.aiRTrigActionPanelLeft[3]:=0;
ptrConfigPage^.aiRTrigActionPanelLeft[4]:=0;
ptrConfigPage^.aiRTrigActionPanelLeft[5]:=11000 + gT_PageNumber.iAutoMode_Parameter;		(* Parameter Page *)
ptrConfigPage^.aiRTrigActionPanelRight[1]:=10000 + gT_PageNumber.iAutoMode_Process;
ptrConfigPage^.aiRTrigActionPanelRight[2]:=10000 + gT_PageNumber.iAutoMode_ProcessValue1;
ptrConfigPage^.aiRTrigActionPanelRight[3]:=10000 + gT_PageNumber.iAutoMode_ProcessValue2;
ptrConfigPage^.aiRTrigActionPanelRight[4]:=10000 + gT_PageNumber.iAutoMode_PartQuality;
ptrConfigPage^.aiRTrigActionPanelRight[5]:=104;		(* Meldungsfenster Öffnen *)
ptrConfigPage^.aiFTrigActionPanelRight[1]:=0;
ptrConfigPage^.aiFTrigActionPanelRight[2]:=0;
ptrConfigPage^.aiFTrigActionPanelRight[3]:=0;
ptrConfigPage^.aiFTrigActionPanelRight[4]:=0;
ptrConfigPage^.aiFTrigActionPanelRight[5]:=0;
ptrConfigPage^.aiRTrigActionFunctionPanel[1]:=150;	(* Löschen des Prozesszustandspeicher *)
ptrConfigPage^.aiRTrigActionFunctionPanel[2]:=0;
ptrConfigPage^.aiRTrigActionFunctionPanel[3]:=0;
ptrConfigPage^.aiRTrigActionFunctionPanel[4]:=0;
ptrConfigPage^.aiRTrigActionFunctionPanel[5]:=0;
ptrConfigPage^.aiRTrigActionFunctionPanel[6]:=0;
ptrConfigPage^.aiRTrigActionFunctionPanel[7]:=0;
ptrConfigPage^.aiRTrigActionFunctionPanel[8]:=0;
ptrConfigPage^.aiRTrigActionFunctionPanel[9]:=0;
ptrConfigPage^.aiRTrigActionFunctionPanel[10]:=0;
ptrConfigPage^.aiRTrigActionFunctionPanel[11]:=0;
ptrConfigPage^.aiRTrigActionFunctionPanel[12]:=0;
TaskBar_NormalMode;
ptrConfigPage^.xMaskBtStart:=TRUE;
ptrConfigPage^.xMaskBtStop:=TRUE;
END_ACTION
ACTION Page_020_AutoMode_Referencing:
(* QVis page 20, AutoMode Referencing *)
iIndexPage:=gT_PageNumber.iAutoMode_Referencing;
iPageNumber:=iPageNumber+1;
T_Visu.T_PageIndex[iIndexPage].iIndexConfigPage:=iPageNumber;
ptrConfigPage:=ADR(T_Visu.T_ConfigPage[T_Visu.T_PageIndex[iIndexPage].iIndexConfigPage]);
ptrConfigPage^.sName:='AutoMode Referencing';
ptrConfigPage^.wMaskBtPanelLeft:=16#18;	(* Parameter *)
ptrConfigPage^.wMaskBtPanelRight:=16#0;
ptrConfigPage^.wMaskFunctionPanel:=16#1;
(* Process mask *)
ptrConfigPage^.wMaskProcBtPanelLeft:=16#F;
ptrConfigPage^.wMaskProcBtPanelRight:=16#0;
ptrConfigPage^.wMaskProcFunctionPanel:=16#0;
(* Button edge action *)
ptrConfigPage^.aiRTrigActionPanelLeft[1]:=0;
ptrConfigPage^.aiRTrigActionPanelLeft[2]:=0;
ptrConfigPage^.aiRTrigActionPanelLeft[3]:=0;
ptrConfigPage^.aiRTrigActionPanelLeft[4]:=0;
ptrConfigPage^.aiRTrigActionPanelLeft[5]:=11000 + gT_PageNumber.iAutoMode_Parameter;		(* Parameter Page *)
ptrConfigPage^.aiRTrigActionPanelRight[1]:=0;
ptrConfigPage^.aiRTrigActionPanelRight[2]:=0;
ptrConfigPage^.aiRTrigActionPanelRight[3]:=0;
ptrConfigPage^.aiRTrigActionPanelRight[4]:=0;
ptrConfigPage^.aiRTrigActionPanelRight[5]:=0;
ptrConfigPage^.aiFTrigActionPanelRight[1]:=0;
ptrConfigPage^.aiFTrigActionPanelRight[2]:=0;
ptrConfigPage^.aiFTrigActionPanelRight[3]:=0;
ptrConfigPage^.aiFTrigActionPanelRight[4]:=0;
ptrConfigPage^.aiFTrigActionPanelRight[5]:=0;
ptrConfigPage^.aiRTrigActionFunctionPanel[1]:=198;	(* Spindelkalibrierung EIN/AUS St1/St3 *)
ptrConfigPage^.aiRTrigActionFunctionPanel[2]:=0;
ptrConfigPage^.aiRTrigActionFunctionPanel[3]:=0;
ptrConfigPage^.aiRTrigActionFunctionPanel[4]:=0;
ptrConfigPage^.aiRTrigActionFunctionPanel[5]:=0;
ptrConfigPage^.aiRTrigActionFunctionPanel[6]:=0;
ptrConfigPage^.aiRTrigActionFunctionPanel[7]:=0;
ptrConfigPage^.aiRTrigActionFunctionPanel[8]:=0;
ptrConfigPage^.aiRTrigActionFunctionPanel[9]:=0;
ptrConfigPage^.aiRTrigActionFunctionPanel[10]:=0;
ptrConfigPage^.aiRTrigActionFunctionPanel[11]:=0;
ptrConfigPage^.aiRTrigActionFunctionPanel[12]:=0;
TaskBar_NormalMode;
ptrConfigPage^.xMaskBtStart:=TRUE;
ptrConfigPage^.xMaskBtStop:=TRUE;
END_ACTION
ACTION Page_030_AutoMode_Profile:
(* QVis page 30, AutoMode Profile *)
iIndexPage:=gT_PageNumber.iAutoMode_Profile;
iPageNumber:=iPageNumber+1;
T_Visu.T_PageIndex[iIndexPage].iIndexConfigPage:=iPageNumber;
ptrConfigPage:=ADR(T_Visu.T_ConfigPage[T_Visu.T_PageIndex[iIndexPage].iIndexConfigPage]);
ptrConfigPage^.sName:='AutoMode Profile';
ptrConfigPage^.wMaskBtPanelLeft:=16#18;	(* Parameter *)
ptrConfigPage^.wMaskBtPanelRight:=16#20;	(* Profil laden *)
ptrConfigPage^.wMaskFunctionPanel:=16#0;
(* Process mask *)
ptrConfigPage^.wMaskProcBtPanelLeft:=16#F;
ptrConfigPage^.wMaskProcBtPanelRight:=16#0;
ptrConfigPage^.wMaskProcFunctionPanel:=16#0;
(* Button edge action *)
ptrConfigPage^.aiRTrigActionPanelLeft[1]:=0;
ptrConfigPage^.aiRTrigActionPanelLeft[2]:=0;
ptrConfigPage^.aiRTrigActionPanelLeft[3]:=0;
ptrConfigPage^.aiRTrigActionPanelLeft[4]:=0;
ptrConfigPage^.aiRTrigActionPanelLeft[5]:=11000 + gT_PageNumber.iAutoMode_Parameter;		(* Parameter Page *)
ptrConfigPage^.aiRTrigActionPanelRight[1]:=1003;		(* Profil laden *)
ptrConfigPage^.aiRTrigActionPanelRight[2]:=0;
ptrConfigPage^.aiRTrigActionPanelRight[3]:=0;
ptrConfigPage^.aiRTrigActionPanelRight[4]:=0;
ptrConfigPage^.aiRTrigActionPanelRight[5]:=0;
ptrConfigPage^.aiFTrigActionPanelRight[1]:=0;
ptrConfigPage^.aiFTrigActionPanelRight[2]:=0;
ptrConfigPage^.aiFTrigActionPanelRight[3]:=0;
ptrConfigPage^.aiFTrigActionPanelRight[4]:=0;
ptrConfigPage^.aiFTrigActionPanelRight[5]:=0;
ptrConfigPage^.aiRTrigActionFunctionPanel[1]:=0;
ptrConfigPage^.aiRTrigActionFunctionPanel[2]:=0;
ptrConfigPage^.aiRTrigActionFunctionPanel[3]:=0;
ptrConfigPage^.aiRTrigActionFunctionPanel[4]:=0;
ptrConfigPage^.aiRTrigActionFunctionPanel[5]:=0;
ptrConfigPage^.aiRTrigActionFunctionPanel[6]:=0;
ptrConfigPage^.aiRTrigActionFunctionPanel[7]:=0;
ptrConfigPage^.aiRTrigActionFunctionPanel[8]:=0;
ptrConfigPage^.aiRTrigActionFunctionPanel[9]:=0;
ptrConfigPage^.aiRTrigActionFunctionPanel[10]:=0;
ptrConfigPage^.aiRTrigActionFunctionPanel[11]:=0;
ptrConfigPage^.aiRTrigActionFunctionPanel[12]:=0;
TaskBar_NormalMode;
ptrConfigPage^.xMaskBtStart:=FALSE;
ptrConfigPage^.xMaskBtStop:=TRUE;
END_ACTION
ACTION Page_040_AutoMode_ToolChange:
(* QVis page 40, AutoMode ToolChange *)
iIndexPage:=gT_PageNumber.iAutoMode_ToolChange;
iPageNumber:=iPageNumber+1;
T_Visu.T_PageIndex[iIndexPage].iIndexConfigPage:=iPageNumber;
ptrConfigPage:=ADR(T_Visu.T_ConfigPage[T_Visu.T_PageIndex[iIndexPage].iIndexConfigPage]);
ptrConfigPage^.sName:='AutoMode ToolChange';
ptrConfigPage^.wMaskBtPanelLeft:=16#18;	(* Parameter *)
ptrConfigPage^.wMaskBtPanelRight:=16#E0;
ptrConfigPage^.wMaskFunctionPanel:=16#7F;	(* F1,F2,F3,F4,F5F6 *)
(* Process mask *)
ptrConfigPage^.wMaskProcBtPanelLeft:=16#F;
ptrConfigPage^.wMaskProcBtPanelRight:=16#E0;
ptrConfigPage^.wMaskProcFunctionPanel:=16#18;
(* Button edge action *)
ptrConfigPage^.aiRTrigActionPanelLeft[1]:=0;
ptrConfigPage^.aiRTrigActionPanelLeft[2]:=0;
ptrConfigPage^.aiRTrigActionPanelLeft[3]:=0;
ptrConfigPage^.aiRTrigActionPanelLeft[4]:=0;
ptrConfigPage^.aiRTrigActionPanelLeft[5]:=11000 + gT_PageNumber.iAutoMode_Parameter;		(* Parameter Page *)
ptrConfigPage^.aiRTrigActionPanelRight[1]:=10000 + gT_PageNumber.iAutoMode_ToolChange;
ptrConfigPage^.aiRTrigActionPanelRight[2]:=10000 + gT_PageNumber.iAutoMode_UserLevel;
ptrConfigPage^.aiRTrigActionPanelRight[3]:=10000 + gT_PageNumber.iAutoMode_Language;
ptrConfigPage^.aiRTrigActionPanelRight[4]:=0;
ptrConfigPage^.aiRTrigActionPanelRight[5]:=0;
ptrConfigPage^.aiFTrigActionPanelRight[1]:=0;
ptrConfigPage^.aiFTrigActionPanelRight[2]:=0;
ptrConfigPage^.aiFTrigActionPanelRight[3]:=0;
ptrConfigPage^.aiFTrigActionPanelRight[4]:=0;
ptrConfigPage^.aiFTrigActionPanelRight[5]:=0;
ptrConfigPage^.aiRTrigActionFunctionPanel[1]:=115;		(* Reset St1 WzWechsel-->With Operator Level *)
ptrConfigPage^.aiRTrigActionFunctionPanel[2]:=116;		(* Z Achse auf WzWechsel Pos setzen *)
ptrConfigPage^.aiRTrigActionFunctionPanel[3]:=117;		(* Z Achse auf LadePos setzen *)
ptrConfigPage^.aiRTrigActionFunctionPanel[4]:=113;		(* Umschalten Z Ink Wert für Bearbeitung *)
ptrConfigPage^.aiRTrigActionFunctionPanel[5]:=114;		(* Umschalten Z Ink Wert für Zentrierung *)
ptrConfigPage^.aiRTrigActionFunctionPanel[6]:=118;		(* Speichern Z EndPos Berechnet *)
ptrConfigPage^.aiRTrigActionFunctionPanel[7]:=0;
ptrConfigPage^.aiRTrigActionFunctionPanel[8]:=0;
ptrConfigPage^.aiRTrigActionFunctionPanel[9]:=0;
ptrConfigPage^.aiRTrigActionFunctionPanel[10]:=0;
ptrConfigPage^.aiRTrigActionFunctionPanel[11]:=0;
ptrConfigPage^.aiRTrigActionFunctionPanel[12]:=0;
TaskBar_NormalMode;
ptrConfigPage^.xMaskBtStart:=FALSE;
ptrConfigPage^.xMaskBtStop:=TRUE;
END_ACTION
ACTION Page_041_AutoMode_UserLevel:
(* QVis page 41, AutoMode UserLevel *)
iIndexPage:=gT_PageNumber.iAutoMode_UserLevel;
iPageNumber:=iPageNumber+1;
T_Visu.T_PageIndex[iIndexPage].iIndexConfigPage:=iPageNumber;
ptrConfigPage:=ADR(T_Visu.T_ConfigPage[T_Visu.T_PageIndex[iIndexPage].iIndexConfigPage]);
ptrConfigPage^.sName:='AutoMode UserLevel';
ptrConfigPage^.wMaskBtPanelLeft:=16#18;	(* Parameter *)
ptrConfigPage^.wMaskBtPanelRight:=16#3E0;
ptrConfigPage^.wMaskFunctionPanel:=16#0;
(* Process mask *)
ptrConfigPage^.wMaskProcBtPanelLeft:=16#F;
ptrConfigPage^.wMaskProcBtPanelRight:=16#3E0;
ptrConfigPage^.wMaskProcFunctionPanel:=16#0;
(* Button edge action *)
ptrConfigPage^.aiRTrigActionPanelLeft[1]:=0;
ptrConfigPage^.aiRTrigActionPanelLeft[2]:=0;
ptrConfigPage^.aiRTrigActionPanelLeft[3]:=0;
ptrConfigPage^.aiRTrigActionPanelLeft[4]:=0;
ptrConfigPage^.aiRTrigActionPanelLeft[5]:=11000 + gT_PageNumber.iAutoMode_Parameter;		(* Parameter Page *)
ptrConfigPage^.aiRTrigActionPanelRight[1]:=10000 + gT_PageNumber.iAutoMode_ToolChange;
ptrConfigPage^.aiRTrigActionPanelRight[2]:=10000 + gT_PageNumber.iAutoMode_UserLevel;
ptrConfigPage^.aiRTrigActionPanelRight[3]:=10000 + gT_PageNumber.iAutoMode_Language;
ptrConfigPage^.aiRTrigActionPanelRight[4]:=0;
ptrConfigPage^.aiRTrigActionPanelRight[5]:=0;
ptrConfigPage^.aiFTrigActionPanelRight[1]:=0;
ptrConfigPage^.aiFTrigActionPanelRight[2]:=0;
ptrConfigPage^.aiFTrigActionPanelRight[3]:=0;
ptrConfigPage^.aiFTrigActionPanelRight[4]:=0;
ptrConfigPage^.aiFTrigActionPanelRight[5]:=0;
ptrConfigPage^.aiRTrigActionFunctionPanel[1]:=110;	(* Wenn OperatorLevel aktiv ist, dann wird diese Funktion freigeschaltet für das Passwort ändern zu können *)
ptrConfigPage^.aiRTrigActionFunctionPanel[2]:=0;
ptrConfigPage^.aiRTrigActionFunctionPanel[3]:=0;
ptrConfigPage^.aiRTrigActionFunctionPanel[4]:=0;
ptrConfigPage^.aiRTrigActionFunctionPanel[5]:=0;
ptrConfigPage^.aiRTrigActionFunctionPanel[6]:=0;
ptrConfigPage^.aiRTrigActionFunctionPanel[7]:=0;
ptrConfigPage^.aiRTrigActionFunctionPanel[8]:=0;
ptrConfigPage^.aiRTrigActionFunctionPanel[9]:=0;
ptrConfigPage^.aiRTrigActionFunctionPanel[10]:=0;
ptrConfigPage^.aiRTrigActionFunctionPanel[11]:=0;
ptrConfigPage^.aiRTrigActionFunctionPanel[12]:=0;
TaskBar_NormalMode;
ptrConfigPage^.xMaskBtStart:=FALSE;
ptrConfigPage^.xMaskBtStop:=TRUE;
END_ACTION
ACTION Page_042_AutoMode_Language:
(* QVis page 42, AutoMode Language *)
iIndexPage:=gT_PageNumber.iAutoMode_Language;
iPageNumber:=iPageNumber+1;
T_Visu.T_PageIndex[iIndexPage].iIndexConfigPage:=iPageNumber;
ptrConfigPage:=ADR(T_Visu.T_ConfigPage[T_Visu.T_PageIndex[iIndexPage].iIndexConfigPage]);
ptrConfigPage^.sName:='AutoMode Language';
ptrConfigPage^.wMaskBtPanelLeft:=16#18;	(* Parameter *)
ptrConfigPage^.wMaskBtPanelRight:=16#3E0;
ptrConfigPage^.wMaskFunctionPanel:=16#0;
(* Process mask *)
ptrConfigPage^.wMaskProcBtPanelLeft:=16#F;
ptrConfigPage^.wMaskProcBtPanelRight:=16#3E0;
ptrConfigPage^.wMaskProcFunctionPanel:=16#0;
(* Button edge action *)
ptrConfigPage^.aiRTrigActionPanelLeft[1]:=0;
ptrConfigPage^.aiRTrigActionPanelLeft[2]:=0;
ptrConfigPage^.aiRTrigActionPanelLeft[3]:=0;
ptrConfigPage^.aiRTrigActionPanelLeft[4]:=0;
ptrConfigPage^.aiRTrigActionPanelLeft[5]:=11000 + gT_PageNumber.iAutoMode_Parameter;		(* Parameter Page *)
ptrConfigPage^.aiRTrigActionPanelRight[1]:=10000 + gT_PageNumber.iAutoMode_ToolChange;
ptrConfigPage^.aiRTrigActionPanelRight[2]:=10000 + gT_PageNumber.iAutoMode_UserLevel;
ptrConfigPage^.aiRTrigActionPanelRight[3]:=10000 + gT_PageNumber.iAutoMode_Language;
ptrConfigPage^.aiRTrigActionPanelRight[4]:=0;
ptrConfigPage^.aiRTrigActionPanelRight[5]:=0;
ptrConfigPage^.aiFTrigActionPanelRight[1]:=0;
ptrConfigPage^.aiFTrigActionPanelRight[2]:=0;
ptrConfigPage^.aiFTrigActionPanelRight[3]:=0;
ptrConfigPage^.aiFTrigActionPanelRight[4]:=0;
ptrConfigPage^.aiFTrigActionPanelRight[5]:=0;
ptrConfigPage^.aiRTrigActionFunctionPanel[1]:=0;
ptrConfigPage^.aiRTrigActionFunctionPanel[2]:=0;
ptrConfigPage^.aiRTrigActionFunctionPanel[3]:=0;
ptrConfigPage^.aiRTrigActionFunctionPanel[4]:=0;
ptrConfigPage^.aiRTrigActionFunctionPanel[5]:=0;
ptrConfigPage^.aiRTrigActionFunctionPanel[6]:=0;
ptrConfigPage^.aiRTrigActionFunctionPanel[7]:=0;
ptrConfigPage^.aiRTrigActionFunctionPanel[8]:=0;
ptrConfigPage^.aiRTrigActionFunctionPanel[9]:=0;
ptrConfigPage^.aiRTrigActionFunctionPanel[10]:=0;
ptrConfigPage^.aiRTrigActionFunctionPanel[11]:=0;
ptrConfigPage^.aiRTrigActionFunctionPanel[12]:=0;
TaskBar_NormalMode;
ptrConfigPage^.xMaskBtStart:=FALSE;
ptrConfigPage^.xMaskBtStop:=TRUE;
END_ACTION
ACTION Page_050_AutoMode_WPCounter:
(* QVis page 50, AutoMode WPCounter *)
iIndexPage:=gT_PageNumber.iAutoMode_WPCounter;
iPageNumber:=iPageNumber+1;
T_Visu.T_PageIndex[iIndexPage].iIndexConfigPage:=iPageNumber;
ptrConfigPage:=ADR(T_Visu.T_ConfigPage[T_Visu.T_PageIndex[iIndexPage].iIndexConfigPage]);
ptrConfigPage^.sName:='AutoMode WPCounter';
ptrConfigPage^.wMaskBtPanelLeft:=16#18;	(* Parameter *)
ptrConfigPage^.wMaskBtPanelRight:=16#1E0;
ptrConfigPage^.wMaskFunctionPanel:=16#0;
(* Process mask *)
ptrConfigPage^.wMaskProcBtPanelLeft:=16#F;
ptrConfigPage^.wMaskProcBtPanelRight:=16#1E0;
ptrConfigPage^.wMaskProcFunctionPanel:=16#0;
(* Button edge action *)
ptrConfigPage^.aiRTrigActionPanelLeft[1]:=0;
ptrConfigPage^.aiRTrigActionPanelLeft[2]:=0;
ptrConfigPage^.aiRTrigActionPanelLeft[3]:=0;
ptrConfigPage^.aiRTrigActionPanelLeft[4]:=0;
ptrConfigPage^.aiRTrigActionPanelLeft[5]:=11000 + gT_PageNumber.iAutoMode_Parameter;		(* Parameter Page *)
ptrConfigPage^.aiRTrigActionPanelRight[1]:=10000 + gT_PageNumber.iAutoMode_WPCounter;
ptrConfigPage^.aiRTrigActionPanelRight[2]:=10000 + gT_PageNumber.iAutoMode_LampTest;
ptrConfigPage^.aiRTrigActionPanelRight[3]:=10000 + gT_PageNumber.iAutoMode_SafetyCheck;
ptrConfigPage^.aiRTrigActionPanelRight[4]:=10000 + gT_PageNumber.iAutoMode_SysInfo;
ptrConfigPage^.aiRTrigActionPanelRight[5]:=0;
ptrConfigPage^.aiFTrigActionPanelRight[1]:=0;
ptrConfigPage^.aiFTrigActionPanelRight[2]:=0;
ptrConfigPage^.aiFTrigActionPanelRight[3]:=0;
ptrConfigPage^.aiFTrigActionPanelRight[4]:=0;
ptrConfigPage^.aiFTrigActionPanelRight[5]:=0;
ptrConfigPage^.aiRTrigActionFunctionPanel[1]:=0;
ptrConfigPage^.aiRTrigActionFunctionPanel[2]:=0;
ptrConfigPage^.aiRTrigActionFunctionPanel[3]:=0;
ptrConfigPage^.aiRTrigActionFunctionPanel[4]:=0;
ptrConfigPage^.aiRTrigActionFunctionPanel[5]:=0;
ptrConfigPage^.aiRTrigActionFunctionPanel[6]:=0;
ptrConfigPage^.aiRTrigActionFunctionPanel[7]:=0;
ptrConfigPage^.aiRTrigActionFunctionPanel[8]:=0;
ptrConfigPage^.aiRTrigActionFunctionPanel[9]:=0;
ptrConfigPage^.aiRTrigActionFunctionPanel[10]:=0;
ptrConfigPage^.aiRTrigActionFunctionPanel[11]:=0;
ptrConfigPage^.aiRTrigActionFunctionPanel[12]:=0;
TaskBar_NormalMode;
ptrConfigPage^.xMaskBtStart:=FALSE;
ptrConfigPage^.xMaskBtStop:=TRUE;
END_ACTION
ACTION Page_051_AutoMode_LampTest:
(* QVis page 51, AutoMode LampTest *)
iIndexPage:=gT_PageNumber.iAutoMode_LampTest;
iPageNumber:=iPageNumber+1;
T_Visu.T_PageIndex[iIndexPage].iIndexConfigPage:=iPageNumber;
ptrConfigPage:=ADR(T_Visu.T_ConfigPage[T_Visu.T_PageIndex[iIndexPage].iIndexConfigPage]);
ptrConfigPage^.sName:='AutoMode LampTest';
ptrConfigPage^.wMaskBtPanelLeft:=16#10;	(* Parameter *)
ptrConfigPage^.wMaskBtPanelRight:=16#1E0;
ptrConfigPage^.wMaskFunctionPanel:=16#7;
(* Process mask *)
ptrConfigPage^.wMaskProcBtPanelLeft:=16#F;
ptrConfigPage^.wMaskProcBtPanelRight:=16#1E0;
ptrConfigPage^.wMaskProcFunctionPanel:=16#0;
(* Button edge action *)
ptrConfigPage^.aiRTrigActionPanelLeft[1]:=0;
ptrConfigPage^.aiRTrigActionPanelLeft[2]:=0;
ptrConfigPage^.aiRTrigActionPanelLeft[3]:=0;
ptrConfigPage^.aiRTrigActionPanelLeft[4]:=0;
ptrConfigPage^.aiRTrigActionPanelLeft[5]:=11000 + gT_PageNumber.iAutoMode_Parameter;		(* Parameter Page *)
ptrConfigPage^.aiRTrigActionPanelRight[1]:=10000 + gT_PageNumber.iAutoMode_WPCounter;
ptrConfigPage^.aiRTrigActionPanelRight[2]:=10000 + gT_PageNumber.iAutoMode_LampTest;
ptrConfigPage^.aiRTrigActionPanelRight[3]:=10000 + gT_PageNumber.iAutoMode_SafetyCheck;
ptrConfigPage^.aiRTrigActionPanelRight[4]:=10000 + gT_PageNumber.iAutoMode_SysInfo;
ptrConfigPage^.aiRTrigActionPanelRight[5]:=0;
ptrConfigPage^.aiFTrigActionPanelRight[1]:=0;
ptrConfigPage^.aiFTrigActionPanelRight[2]:=0;
ptrConfigPage^.aiFTrigActionPanelRight[3]:=0;
ptrConfigPage^.aiFTrigActionPanelRight[4]:=0;
ptrConfigPage^.aiFTrigActionPanelRight[5]:=0;
ptrConfigPage^.aiRTrigActionFunctionPanel[1]:=100;		(* Lampen EIN/AUS *)
ptrConfigPage^.aiRTrigActionFunctionPanel[2]:=101;		(* Lampen Blinken *)
ptrConfigPage^.aiRTrigActionFunctionPanel[3]:=102;		(* Lampen Test *)
ptrConfigPage^.aiRTrigActionFunctionPanel[4]:=0;
ptrConfigPage^.aiRTrigActionFunctionPanel[5]:=0;
ptrConfigPage^.aiRTrigActionFunctionPanel[6]:=0;
ptrConfigPage^.aiRTrigActionFunctionPanel[7]:=0;
ptrConfigPage^.aiRTrigActionFunctionPanel[8]:=0;
ptrConfigPage^.aiRTrigActionFunctionPanel[9]:=0;
ptrConfigPage^.aiRTrigActionFunctionPanel[10]:=0;
ptrConfigPage^.aiRTrigActionFunctionPanel[11]:=0;
ptrConfigPage^.aiRTrigActionFunctionPanel[12]:=0;
TaskBar_NormalMode;
ptrConfigPage^.xMaskBtStart:=FALSE;
ptrConfigPage^.xMaskBtStop:=TRUE;
END_ACTION
ACTION Page_052_AutoMode_SafetyCheck:
(* QVis page 52, AutoMode SafetyCheck *)
iIndexPage:=gT_PageNumber.iAutoMode_SafetyCheck;
iPageNumber:=iPageNumber+1;
T_Visu.T_PageIndex[iIndexPage].iIndexConfigPage:=iPageNumber;
ptrConfigPage:=ADR(T_Visu.T_ConfigPage[T_Visu.T_PageIndex[iIndexPage].iIndexConfigPage]);
ptrConfigPage^.sName:='AutoMode SafetyCheck';
ptrConfigPage^.wMaskBtPanelLeft:=16#18;	(* Parameter *)
ptrConfigPage^.wMaskBtPanelRight:=16#1E0;
ptrConfigPage^.wMaskFunctionPanel:=16#1;	(* F1 *)
(* Process mask *)
ptrConfigPage^.wMaskProcBtPanelLeft:=16#F;
ptrConfigPage^.wMaskProcBtPanelRight:=16#1E0;
ptrConfigPage^.wMaskProcFunctionPanel:=16#0;
(* Button edge action *)
ptrConfigPage^.aiRTrigActionPanelLeft[1]:=0;
ptrConfigPage^.aiRTrigActionPanelLeft[2]:=0;
ptrConfigPage^.aiRTrigActionPanelLeft[3]:=0;
ptrConfigPage^.aiRTrigActionPanelLeft[4]:=0;
ptrConfigPage^.aiRTrigActionPanelLeft[5]:=11000 + gT_PageNumber.iAutoMode_Parameter;		(* Parameter Page *)
ptrConfigPage^.aiRTrigActionPanelRight[1]:=10000 + gT_PageNumber.iAutoMode_WPCounter;
ptrConfigPage^.aiRTrigActionPanelRight[2]:=10000 + gT_PageNumber.iAutoMode_LampTest;
ptrConfigPage^.aiRTrigActionPanelRight[3]:=10000 + gT_PageNumber.iAutoMode_SafetyCheck;
ptrConfigPage^.aiRTrigActionPanelRight[4]:=10000 + gT_PageNumber.iAutoMode_SysInfo;
ptrConfigPage^.aiRTrigActionPanelRight[5]:=0;
ptrConfigPage^.aiFTrigActionPanelRight[1]:=0;
ptrConfigPage^.aiFTrigActionPanelRight[2]:=0;
ptrConfigPage^.aiFTrigActionPanelRight[3]:=0;
ptrConfigPage^.aiFTrigActionPanelRight[4]:=0;
ptrConfigPage^.aiFTrigActionPanelRight[5]:=0;
ptrConfigPage^.aiRTrigActionFunctionPanel[1]:=105;		(* Maschinen Tür Zuhaltung EIN/AUS *)
ptrConfigPage^.aiRTrigActionFunctionPanel[2]:=0;
ptrConfigPage^.aiRTrigActionFunctionPanel[3]:=0;
ptrConfigPage^.aiRTrigActionFunctionPanel[4]:=0;
ptrConfigPage^.aiRTrigActionFunctionPanel[5]:=0;
ptrConfigPage^.aiRTrigActionFunctionPanel[6]:=0;
ptrConfigPage^.aiRTrigActionFunctionPanel[7]:=0;
ptrConfigPage^.aiRTrigActionFunctionPanel[8]:=0;
ptrConfigPage^.aiRTrigActionFunctionPanel[9]:=0;
ptrConfigPage^.aiRTrigActionFunctionPanel[10]:=0;
ptrConfigPage^.aiRTrigActionFunctionPanel[11]:=0;
ptrConfigPage^.aiRTrigActionFunctionPanel[12]:=0;
TaskBar_NormalMode;
ptrConfigPage^.xMaskBtStart:=FALSE;
ptrConfigPage^.xMaskBtStop:=TRUE;
END_ACTION
ACTION Page_053_AutoMode_SysInfo:
(* QVis page 53, AutoMode SysInfo *)
iIndexPage:=gT_PageNumber.iAutoMode_SysInfo;
iPageNumber:=iPageNumber+1;
T_Visu.T_PageIndex[iIndexPage].iIndexConfigPage:=iPageNumber;
ptrConfigPage:=ADR(T_Visu.T_ConfigPage[T_Visu.T_PageIndex[iIndexPage].iIndexConfigPage]);
ptrConfigPage^.sName:='AutoMode SysInfo';
ptrConfigPage^.wMaskBtPanelLeft:=16#18;	(* Parameter *)
ptrConfigPage^.wMaskBtPanelRight:=16#1E0;
ptrConfigPage^.wMaskFunctionPanel:=16#0;
(* Process mask *)
ptrConfigPage^.wMaskProcBtPanelLeft:=16#F;
ptrConfigPage^.wMaskProcBtPanelRight:=16#1E0;
ptrConfigPage^.wMaskProcFunctionPanel:=16#0;
(* Button edge action *)
ptrConfigPage^.aiRTrigActionPanelLeft[1]:=0;
ptrConfigPage^.aiRTrigActionPanelLeft[2]:=0;
ptrConfigPage^.aiRTrigActionPanelLeft[3]:=0;
ptrConfigPage^.aiRTrigActionPanelLeft[4]:=0;
ptrConfigPage^.aiRTrigActionPanelLeft[5]:=11000 + gT_PageNumber.iAutoMode_Parameter;		(* Parameter Page *)
ptrConfigPage^.aiRTrigActionPanelRight[1]:=10000 + gT_PageNumber.iAutoMode_WPCounter;
ptrConfigPage^.aiRTrigActionPanelRight[2]:=10000 + gT_PageNumber.iAutoMode_LampTest;
ptrConfigPage^.aiRTrigActionPanelRight[3]:=10000 + gT_PageNumber.iAutoMode_SafetyCheck;
ptrConfigPage^.aiRTrigActionPanelRight[4]:=10000 + gT_PageNumber.iAutoMode_SysInfo;
ptrConfigPage^.aiRTrigActionPanelRight[5]:=0;
ptrConfigPage^.aiFTrigActionPanelRight[1]:=0;
ptrConfigPage^.aiFTrigActionPanelRight[2]:=0;
ptrConfigPage^.aiFTrigActionPanelRight[3]:=0;
ptrConfigPage^.aiFTrigActionPanelRight[4]:=0;
ptrConfigPage^.aiFTrigActionPanelRight[5]:=0;
ptrConfigPage^.aiRTrigActionFunctionPanel[1]:=0;
ptrConfigPage^.aiRTrigActionFunctionPanel[2]:=0;
ptrConfigPage^.aiRTrigActionFunctionPanel[3]:=0;
ptrConfigPage^.aiRTrigActionFunctionPanel[4]:=0;
ptrConfigPage^.aiRTrigActionFunctionPanel[5]:=0;
ptrConfigPage^.aiRTrigActionFunctionPanel[6]:=0;
ptrConfigPage^.aiRTrigActionFunctionPanel[7]:=0;
ptrConfigPage^.aiRTrigActionFunctionPanel[8]:=0;
ptrConfigPage^.aiRTrigActionFunctionPanel[9]:=0;
ptrConfigPage^.aiRTrigActionFunctionPanel[10]:=0;
ptrConfigPage^.aiRTrigActionFunctionPanel[11]:=0;
ptrConfigPage^.aiRTrigActionFunctionPanel[12]:=0;
TaskBar_NormalMode;
ptrConfigPage^.xMaskBtStart:=FALSE;
ptrConfigPage^.xMaskBtStop:=TRUE;
END_ACTION
ACTION Page_060_AutoMode_ErrorList:
(* QVis page 60, AutoMode ErrorList *)
iIndexPage:=gT_PageNumber.iAutoMode_ErrorList;
iPageNumber:=iPageNumber+1;
T_Visu.T_PageIndex[iIndexPage].iIndexConfigPage:=iPageNumber;
ptrConfigPage:=ADR(T_Visu.T_ConfigPage[T_Visu.T_PageIndex[iIndexPage].iIndexConfigPage]);
ptrConfigPage^.sName:='AutoMode ErrorList';
ptrConfigPage^.wMaskBtPanelLeft:=16#18;	(* Parameter *)
ptrConfigPage^.wMaskBtPanelRight:=16#60;	(* Reset Fehler, Löschen Fehlerliste *)
ptrConfigPage^.wMaskFunctionPanel:=16#0;
(* Process mask *)
ptrConfigPage^.wMaskProcBtPanelLeft:=16#F;
ptrConfigPage^.wMaskProcBtPanelRight:=16#0;
ptrConfigPage^.wMaskProcFunctionPanel:=16#0;
(* Button edge action *)
ptrConfigPage^.aiRTrigActionPanelLeft[1]:=0;
ptrConfigPage^.aiRTrigActionPanelLeft[2]:=0;
ptrConfigPage^.aiRTrigActionPanelLeft[3]:=0;
ptrConfigPage^.aiRTrigActionPanelLeft[4]:=0;
ptrConfigPage^.aiRTrigActionPanelLeft[5]:=11000 + gT_PageNumber.iAutoMode_Parameter;		(* Parameter Page *)
ptrConfigPage^.aiRTrigActionPanelRight[1]:=99;		(* Reset Fehler *)
ptrConfigPage^.aiRTrigActionPanelRight[2]:=97;		(* Löschen Fehlerliste *)
ptrConfigPage^.aiRTrigActionPanelRight[3]:=0;
ptrConfigPage^.aiRTrigActionPanelRight[4]:=0;
ptrConfigPage^.aiRTrigActionPanelRight[5]:=0;
ptrConfigPage^.aiFTrigActionPanelRight[1]:=0;
ptrConfigPage^.aiFTrigActionPanelRight[2]:=0;
ptrConfigPage^.aiFTrigActionPanelRight[3]:=0;
ptrConfigPage^.aiFTrigActionPanelRight[4]:=0;
ptrConfigPage^.aiFTrigActionPanelRight[5]:=0;
ptrConfigPage^.aiRTrigActionFunctionPanel[1]:=0;
ptrConfigPage^.aiRTrigActionFunctionPanel[2]:=0;
ptrConfigPage^.aiRTrigActionFunctionPanel[3]:=0;
ptrConfigPage^.aiRTrigActionFunctionPanel[4]:=0;
ptrConfigPage^.aiRTrigActionFunctionPanel[5]:=0;
ptrConfigPage^.aiRTrigActionFunctionPanel[6]:=0;
ptrConfigPage^.aiRTrigActionFunctionPanel[7]:=0;
ptrConfigPage^.aiRTrigActionFunctionPanel[8]:=0;
ptrConfigPage^.aiRTrigActionFunctionPanel[9]:=0;
ptrConfigPage^.aiRTrigActionFunctionPanel[10]:=0;
ptrConfigPage^.aiRTrigActionFunctionPanel[11]:=0;
ptrConfigPage^.aiRTrigActionFunctionPanel[12]:=0;
TaskBar_NormalMode;
ptrConfigPage^.xMaskBtStart:=FALSE;
ptrConfigPage^.xMaskBtStop:=TRUE;
END_ACTION
ACTION Page_070_AutoMode_Parameter:
(* QVis page 70, AutoMode Parameter *)
iIndexPage:=gT_PageNumber.iAutoMode_Parameter;
iPageNumber:=iPageNumber+1;
T_Visu.T_PageIndex[iIndexPage].iIndexConfigPage:=iPageNumber;
ptrConfigPage:=ADR(T_Visu.T_ConfigPage[T_Visu.T_PageIndex[iIndexPage].iIndexConfigPage]);
ptrConfigPage^.sName:='AutoMode Parameter';
ptrConfigPage^.wMaskBtPanelLeft:=16#18;	(* Parameter *)
ptrConfigPage^.wMaskBtPanelRight:=16#200;	(* Speichern *)
ptrConfigPage^.wMaskFunctionPanel:=16#0;
(* Process mask *)
ptrConfigPage^.wMaskProcBtPanelLeft:=16#F;
ptrConfigPage^.wMaskProcBtPanelRight:=16#200;	(* Speichern *)
ptrConfigPage^.wMaskProcFunctionPanel:=16#0;
(* Button edge action *)
ptrConfigPage^.aiRTrigActionPanelLeft[1]:=0;
ptrConfigPage^.aiRTrigActionPanelLeft[2]:=0;
ptrConfigPage^.aiRTrigActionPanelLeft[3]:=0;
ptrConfigPage^.aiRTrigActionPanelLeft[4]:=0;
ptrConfigPage^.aiRTrigActionPanelLeft[5]:=5;		(* Parameter OFF-->Previous Page *)
ptrConfigPage^.aiRTrigActionPanelRight[1]:=0;
ptrConfigPage^.aiRTrigActionPanelRight[2]:=0;
ptrConfigPage^.aiRTrigActionPanelRight[3]:=0;
ptrConfigPage^.aiRTrigActionPanelRight[4]:=0;
ptrConfigPage^.aiRTrigActionPanelRight[5]:=1001;		(* Speichern *)
ptrConfigPage^.aiFTrigActionPanelRight[1]:=0;
ptrConfigPage^.aiFTrigActionPanelRight[2]:=0;
ptrConfigPage^.aiFTrigActionPanelRight[3]:=0;
ptrConfigPage^.aiFTrigActionPanelRight[4]:=0;
ptrConfigPage^.aiFTrigActionPanelRight[5]:=0;
ptrConfigPage^.aiRTrigActionFunctionPanel[1]:=0;
ptrConfigPage^.aiRTrigActionFunctionPanel[2]:=0;
ptrConfigPage^.aiRTrigActionFunctionPanel[3]:=0;
ptrConfigPage^.aiRTrigActionFunctionPanel[4]:=0;
ptrConfigPage^.aiRTrigActionFunctionPanel[5]:=0;
ptrConfigPage^.aiRTrigActionFunctionPanel[6]:=0;
ptrConfigPage^.aiRTrigActionFunctionPanel[7]:=0;
ptrConfigPage^.aiRTrigActionFunctionPanel[8]:=0;
ptrConfigPage^.aiRTrigActionFunctionPanel[9]:=0;
ptrConfigPage^.aiRTrigActionFunctionPanel[10]:=0;
ptrConfigPage^.aiRTrigActionFunctionPanel[11]:=0;
ptrConfigPage^.aiRTrigActionFunctionPanel[12]:=0;
TaskBar_NormalMode;
ptrConfigPage^.xMaskBtStart:=FALSE;
ptrConfigPage^.xMaskBtStop:=TRUE;
END_ACTION
ACTION Page_110_HandMode_Process:
(* QVis page 110, HandMode Process *)
iIndexPage:=gT_PageNumber.iHandMode_Process;
iPageNumber:=iPageNumber+1;
T_Visu.T_PageIndex[iIndexPage].iIndexConfigPage:=iPageNumber;
ptrConfigPage:=ADR(T_Visu.T_ConfigPage[T_Visu.T_PageIndex[iIndexPage].iIndexConfigPage]);
ptrConfigPage^.sName:='HandMode Process';
ptrConfigPage^.wMaskBtPanelLeft:=16#19;		(*              1 1001 	SetupModeA, Lampe, Parameter *)
ptrConfigPage^.wMaskBtPanelRight:=16#3E0;		(* 11 1110 0000	Process, WorkParameter, RegulatorPara, OnlineChange, ConfigPosition *)
ptrConfigPage^.wMaskFunctionPanel:=16#0;
(* Process mask *)
ptrConfigPage^.wMaskProcBtPanelLeft:=16#9;		(*              1 1001 	SetupModeA, Lampe *)
ptrConfigPage^.wMaskProcBtPanelRight:=16#3E0;	(* 11 1110 0000	Process, WorkParameter, RegulatorPara, OnlineChange, ConfigPosition *)
ptrConfigPage^.wMaskProcFunctionPanel:=16#0;
(* Button edge action *)
ptrConfigPage^.aiRTrigActionPanelLeft[1]:=0;
ptrConfigPage^.aiRTrigActionPanelLeft[2]:=0;
ptrConfigPage^.aiRTrigActionPanelLeft[3]:=0;
ptrConfigPage^.aiRTrigActionPanelLeft[4]:=0;
ptrConfigPage^.aiRTrigActionPanelLeft[5]:=11000 + gT_PageNumber.iHandMode_Parameter;		(* Parameter Page *)
ptrConfigPage^.aiRTrigActionPanelRight[1]:=10000 + gT_PageNumber.iHandMode_Process;
ptrConfigPage^.aiRTrigActionPanelRight[2]:=10000 + gT_PageNumber.iHandMode_WorkParameter;
ptrConfigPage^.aiRTrigActionPanelRight[3]:=10000 + gT_PageNumber.iHandMode_RegulatorPara;
ptrConfigPage^.aiRTrigActionPanelRight[4]:=10000 + gT_PageNumber.iHandMode_OnlineChange;
ptrConfigPage^.aiRTrigActionPanelRight[5]:=10000 + gT_PageNumber.iHandMode_ConfigPosition;
ptrConfigPage^.aiFTrigActionPanelRight[1]:=0;
ptrConfigPage^.aiFTrigActionPanelRight[2]:=0;
ptrConfigPage^.aiFTrigActionPanelRight[3]:=0;
ptrConfigPage^.aiFTrigActionPanelRight[4]:=0;
ptrConfigPage^.aiFTrigActionPanelRight[5]:=0;
ptrConfigPage^.aiRTrigActionFunctionPanel[1]:=0;
ptrConfigPage^.aiRTrigActionFunctionPanel[2]:=0;
ptrConfigPage^.aiRTrigActionFunctionPanel[3]:=0;
ptrConfigPage^.aiRTrigActionFunctionPanel[4]:=0;
ptrConfigPage^.aiRTrigActionFunctionPanel[5]:=0;
ptrConfigPage^.aiRTrigActionFunctionPanel[6]:=0;
ptrConfigPage^.aiRTrigActionFunctionPanel[7]:=0;
ptrConfigPage^.aiRTrigActionFunctionPanel[8]:=0;
ptrConfigPage^.aiRTrigActionFunctionPanel[9]:=0;
ptrConfigPage^.aiRTrigActionFunctionPanel[10]:=0;
ptrConfigPage^.aiRTrigActionFunctionPanel[11]:=0;
ptrConfigPage^.aiRTrigActionFunctionPanel[12]:=0;
TaskBar_SetupModeA;
ptrConfigPage^.xMaskBtStart:=TRUE;
ptrConfigPage^.xMaskBtStop:=TRUE;
END_ACTION
ACTION Page_111_HandMode_WorkParameter:
(* QVis page 111, HandMode WorkParameter *)
iIndexPage:=gT_PageNumber.iHandMode_WorkParameter;
iPageNumber:=iPageNumber+1;
T_Visu.T_PageIndex[iIndexPage].iIndexConfigPage:=iPageNumber;
ptrConfigPage:=ADR(T_Visu.T_ConfigPage[T_Visu.T_PageIndex[iIndexPage].iIndexConfigPage]);
ptrConfigPage^.sName:='HandMode Work Parameter';
ptrConfigPage^.wMaskBtPanelLeft:=16#19;		(*              1 1001 	SetupModeA, Lampe, Parameter *)
ptrConfigPage^.wMaskBtPanelRight:=16#3E0;		(* 11 1110 0000	Process, WorkParameter, RegulatorPara, OnlineChange, ConfigPosition *)
ptrConfigPage^.wMaskFunctionPanel:=16#0;
(* Process mask *)
ptrConfigPage^.wMaskProcBtPanelLeft:=16#9;		(*              1 1001 	SetupModeA, Lampe *)
ptrConfigPage^.wMaskProcBtPanelRight:=16#3E0;	(* 11 1110 0000	Process, WorkParameter, RegulatorPara, OnlineChange, ConfigPosition *)
ptrConfigPage^.wMaskProcFunctionPanel:=16#0;
(* Button edge action *)
ptrConfigPage^.aiRTrigActionPanelLeft[1]:=0;
ptrConfigPage^.aiRTrigActionPanelLeft[2]:=0;
ptrConfigPage^.aiRTrigActionPanelLeft[3]:=0;
ptrConfigPage^.aiRTrigActionPanelLeft[4]:=0;
ptrConfigPage^.aiRTrigActionPanelLeft[5]:=11000 + gT_PageNumber.iHandMode_Parameter;		(* Parameter Page *)
ptrConfigPage^.aiRTrigActionPanelRight[1]:=10000 + gT_PageNumber.iHandMode_Process;
ptrConfigPage^.aiRTrigActionPanelRight[2]:=10000 + gT_PageNumber.iHandMode_WorkParameter;
ptrConfigPage^.aiRTrigActionPanelRight[3]:=10000 + gT_PageNumber.iHandMode_RegulatorPara;
ptrConfigPage^.aiRTrigActionPanelRight[4]:=10000 + gT_PageNumber.iHandMode_OnlineChange;
ptrConfigPage^.aiRTrigActionPanelRight[5]:=10000 + gT_PageNumber.iHandMode_ConfigPosition;
ptrConfigPage^.aiFTrigActionPanelRight[1]:=0;
ptrConfigPage^.aiFTrigActionPanelRight[2]:=0;
ptrConfigPage^.aiFTrigActionPanelRight[3]:=0;
ptrConfigPage^.aiFTrigActionPanelRight[4]:=0;
ptrConfigPage^.aiFTrigActionPanelRight[5]:=0;
ptrConfigPage^.aiRTrigActionFunctionPanel[1]:=0;
ptrConfigPage^.aiRTrigActionFunctionPanel[2]:=0;
ptrConfigPage^.aiRTrigActionFunctionPanel[3]:=0;
ptrConfigPage^.aiRTrigActionFunctionPanel[4]:=0;
ptrConfigPage^.aiRTrigActionFunctionPanel[5]:=0;
ptrConfigPage^.aiRTrigActionFunctionPanel[6]:=0;
ptrConfigPage^.aiRTrigActionFunctionPanel[7]:=0;
ptrConfigPage^.aiRTrigActionFunctionPanel[8]:=0;
ptrConfigPage^.aiRTrigActionFunctionPanel[9]:=0;
ptrConfigPage^.aiRTrigActionFunctionPanel[10]:=0;
ptrConfigPage^.aiRTrigActionFunctionPanel[11]:=0;
ptrConfigPage^.aiRTrigActionFunctionPanel[12]:=0;
TaskBar_SetupModeA;
ptrConfigPage^.xMaskBtStart:=TRUE;
ptrConfigPage^.xMaskBtStop:=TRUE;
END_ACTION
ACTION Page_112_HandMode_RegulatorPara:
(* QVis page 112, HandMode RegulatorPara *)
iIndexPage:=gT_PageNumber.iHandMode_RegulatorPara;
iPageNumber:=iPageNumber+1;
T_Visu.T_PageIndex[iIndexPage].iIndexConfigPage:=iPageNumber;
ptrConfigPage:=ADR(T_Visu.T_ConfigPage[T_Visu.T_PageIndex[iIndexPage].iIndexConfigPage]);
ptrConfigPage^.sName:='HandMode Regulator Parameter';
ptrConfigPage^.wMaskBtPanelLeft:=16#19;		(*              1 1001 	SetupModeA, Lampe, Parameter *)
ptrConfigPage^.wMaskBtPanelRight:=16#3E0;		(* 11 1110 0000	Process, WorkParameter, RegulatorPara, OnlineChange, ConfigPosition *)
ptrConfigPage^.wMaskFunctionPanel:=16#27;		(* 10 0000 *)
(* Process mask *)
ptrConfigPage^.wMaskProcBtPanelLeft:=16#9;		(*              1 1001 	SetupModeA, Lampe *)
ptrConfigPage^.wMaskProcBtPanelRight:=16#3E0;	(* 11 1110 0000	Process, WorkParameter, RegulatorPara, OnlineChange, ConfigPosition *)
ptrConfigPage^.wMaskProcFunctionPanel:=16#0;
(* Button edge action *)
ptrConfigPage^.aiRTrigActionPanelLeft[1]:=0;
ptrConfigPage^.aiRTrigActionPanelLeft[2]:=0;
ptrConfigPage^.aiRTrigActionPanelLeft[3]:=0;
ptrConfigPage^.aiRTrigActionPanelLeft[4]:=0;
ptrConfigPage^.aiRTrigActionPanelLeft[5]:=11000 + gT_PageNumber.iHandMode_Parameter;		(* Parameter Page *)
ptrConfigPage^.aiRTrigActionPanelRight[1]:=10000 + gT_PageNumber.iHandMode_Process;
ptrConfigPage^.aiRTrigActionPanelRight[2]:=10000 + gT_PageNumber.iHandMode_WorkParameter;
ptrConfigPage^.aiRTrigActionPanelRight[3]:=10000 + gT_PageNumber.iHandMode_RegulatorPara;
ptrConfigPage^.aiRTrigActionPanelRight[4]:=10000 + gT_PageNumber.iHandMode_OnlineChange;
ptrConfigPage^.aiRTrigActionPanelRight[5]:=10000 + gT_PageNumber.iHandMode_ConfigPosition;
ptrConfigPage^.aiFTrigActionPanelRight[1]:=0;
ptrConfigPage^.aiFTrigActionPanelRight[2]:=0;
ptrConfigPage^.aiFTrigActionPanelRight[3]:=0;
ptrConfigPage^.aiFTrigActionPanelRight[4]:=0;
ptrConfigPage^.aiFTrigActionPanelRight[5]:=0;
ptrConfigPage^.aiRTrigActionFunctionPanel[1]:=190;	(* Konventioneller Regler *)
ptrConfigPage^.aiRTrigActionFunctionPanel[2]:=191;	(* Adaptive Voschub Regler *)
ptrConfigPage^.aiRTrigActionFunctionPanel[3]:=192;	(* Konventioneller PD Regler *)
ptrConfigPage^.aiRTrigActionFunctionPanel[4]:=0;
ptrConfigPage^.aiRTrigActionFunctionPanel[5]:=0;
ptrConfigPage^.aiRTrigActionFunctionPanel[6]:=195;	(* Regler Parameter speichern *)
ptrConfigPage^.aiRTrigActionFunctionPanel[7]:=0;
ptrConfigPage^.aiRTrigActionFunctionPanel[8]:=0;
ptrConfigPage^.aiRTrigActionFunctionPanel[9]:=0;
ptrConfigPage^.aiRTrigActionFunctionPanel[10]:=0;
ptrConfigPage^.aiRTrigActionFunctionPanel[11]:=0;
ptrConfigPage^.aiRTrigActionFunctionPanel[12]:=0;
TaskBar_SetupModeA;
ptrConfigPage^.xMaskBtStart:=TRUE;
ptrConfigPage^.xMaskBtStop:=TRUE;
END_ACTION
ACTION Page_113_HandMode_OnlineChange:
(* QVis page 111, HandMode OnlineChange *)
iIndexPage:=gT_PageNumber.iHandMode_OnlineChange;
iPageNumber:=iPageNumber+1;
T_Visu.T_PageIndex[iIndexPage].iIndexConfigPage:=iPageNumber;
ptrConfigPage:=ADR(T_Visu.T_ConfigPage[T_Visu.T_PageIndex[iIndexPage].iIndexConfigPage]);
ptrConfigPage^.sName:='HandMode OnlineChange';
ptrConfigPage^.wMaskBtPanelLeft:=16#19;		(*              1 1001 	SetupModeA, Lampe, Parameter *)
ptrConfigPage^.wMaskBtPanelRight:=16#3E0;		(* 11 1110 0000	Process, WorkParameter, RegulatorPara, OnlineChange, ConfigPosition *)		(* IGS alt: E0;*)
ptrConfigPage^.wMaskFunctionPanel:=16#FFF;	(*configuration by FBQVIS, because page has more than 1 List*)
(* Process mask *)
ptrConfigPage^.wMaskProcBtPanelLeft:=16#9;	(* SetupModeA, Parameter *)
ptrConfigPage^.wMaskProcBtPanelRight:=16#3E0;	(* 11 1110 0000	Process, WorkParameter, RegulatorPara, OnlineChange, ConfigPosition *)		(* IGS alt: E0;*)
ptrConfigPage^.wMaskProcFunctionPanel:=16#0;	(*configuration by FBQVIS, because page has more than 1 List*)
(* Button edge action *)
ptrConfigPage^.aiRTrigActionPanelLeft[1]:=0;
ptrConfigPage^.aiRTrigActionPanelLeft[2]:=0;
ptrConfigPage^.aiRTrigActionPanelLeft[3]:=0;
ptrConfigPage^.aiRTrigActionPanelLeft[4]:=0;
ptrConfigPage^.aiRTrigActionPanelLeft[5]:=11000 + gT_PageNumber.iHandMode_Parameter;		(* Parameter Page *)
ptrConfigPage^.aiRTrigActionPanelRight[1]:=10000 + gT_PageNumber.iHandMode_Process;
ptrConfigPage^.aiRTrigActionPanelRight[2]:=10000 + gT_PageNumber.iHandMode_WorkParameter;
ptrConfigPage^.aiRTrigActionPanelRight[3]:=10000 + gT_PageNumber.iHandMode_RegulatorPara;
ptrConfigPage^.aiRTrigActionPanelRight[4]:=10000 + gT_PageNumber.iHandMode_OnlineChange;
ptrConfigPage^.aiRTrigActionPanelRight[5]:=10000 + gT_PageNumber.iHandMode_ConfigPosition;
ptrConfigPage^.aiFTrigActionPanelRight[1]:=0;
ptrConfigPage^.aiFTrigActionPanelRight[2]:=0;
ptrConfigPage^.aiFTrigActionPanelRight[3]:=0;
ptrConfigPage^.aiFTrigActionPanelRight[4]:=0;
ptrConfigPage^.aiFTrigActionPanelRight[5]:=0;
ptrConfigPage^.aiRTrigActionFunctionPanel[1]:=120;	(*configuration by FBQVIS, because page has more than 1 List*)
ptrConfigPage^.aiRTrigActionFunctionPanel[2]:=126;	(*configuration by FBQVIS, because page has more than 1 List*)
ptrConfigPage^.aiRTrigActionFunctionPanel[3]:=128;	(*configuration by FBQVIS, because page has more than 1 List*)
ptrConfigPage^.aiRTrigActionFunctionPanel[4]:=132;	(*configuration by FBQVIS, because page has more than 1 List*)
ptrConfigPage^.aiRTrigActionFunctionPanel[5]:=130;	(*configuration by FBQVIS, because page has more than 1 List*)
ptrConfigPage^.aiRTrigActionFunctionPanel[6]:=134;	(*configuration by FBQVIS, because page has more than 1 List*)
ptrConfigPage^.aiRTrigActionFunctionPanel[7]:=121;	(*configuration by FBQVIS, because page has more than 1 List*)
ptrConfigPage^.aiRTrigActionFunctionPanel[8]:=127;	(*configuration by FBQVIS, because page has more than 1 List*)
ptrConfigPage^.aiRTrigActionFunctionPanel[9]:=129;	(*configuration by FBQVIS, because page has more than 1 List*)
ptrConfigPage^.aiRTrigActionFunctionPanel[10]:=133;	(*configuration by FBQVIS, because page has more than 1 List*)
ptrConfigPage^.aiRTrigActionFunctionPanel[11]:=131;	(*configuration by FBQVIS, because page has more than 1 List*)
ptrConfigPage^.aiRTrigActionFunctionPanel[12]:=135;	(*configuration by FBQVIS, because page has more than 1 List*)
TaskBar_SetupModeA;
ptrConfigPage^.xMaskBtStart:=TRUE;
ptrConfigPage^.xMaskBtStop:=TRUE;
END_ACTION
ACTION Page_114_HandMode_ConfigPosition:
(* QVis page 112, HandMode Config Position *)
iIndexPage:=gT_PageNumber.iHandMode_ConfigPosition;
iPageNumber:=iPageNumber+1;
T_Visu.T_PageIndex[iIndexPage].iIndexConfigPage:=iPageNumber;
ptrConfigPage:=ADR(T_Visu.T_ConfigPage[T_Visu.T_PageIndex[iIndexPage].iIndexConfigPage]);
ptrConfigPage^.sName:='HandMode Config Position';
ptrConfigPage^.wMaskBtPanelLeft:=16#19;		(*              1 1001 	SetupModeA, Lampe, Parameter *)
ptrConfigPage^.wMaskBtPanelRight:=16#3E0;		(* 11 1110 0000	Process, WorkParameter, RegulatorPara, OnlineChange, ConfigPosition *)		(* IGS alt: E0;*)
ptrConfigPage^.wMaskFunctionPanel:=16#3F;		(* 11 1111 *)
(* Process mask *)
ptrConfigPage^.wMaskProcBtPanelLeft:=16#9;		(*              1 1001 	SetupModeA, Lampe *)
ptrConfigPage^.wMaskProcBtPanelRight:=16#3E0;	(* 11 1110 0000	Process, WorkParameter, RegulatorPara, OnlineChange, ConfigPosition *)		(* IGS alt: E0;*)
ptrConfigPage^.wMaskProcFunctionPanel:=16#F;	(* 00 1111 *)
(* Button edge action *)
ptrConfigPage^.aiRTrigActionPanelLeft[1]:=0;
ptrConfigPage^.aiRTrigActionPanelLeft[2]:=0;
ptrConfigPage^.aiRTrigActionPanelLeft[3]:=0;
ptrConfigPage^.aiRTrigActionPanelLeft[4]:=0;
ptrConfigPage^.aiRTrigActionPanelLeft[5]:=11000 + gT_PageNumber.iHandMode_Parameter;		(* Parameter Page *)
ptrConfigPage^.aiRTrigActionPanelRight[1]:=10000 + gT_PageNumber.iHandMode_Process;
ptrConfigPage^.aiRTrigActionPanelRight[2]:=10000 + gT_PageNumber.iHandMode_WorkParameter;
ptrConfigPage^.aiRTrigActionPanelRight[3]:=10000 + gT_PageNumber.iHandMode_RegulatorPara;
ptrConfigPage^.aiRTrigActionPanelRight[4]:=10000 + gT_PageNumber.iHandMode_OnlineChange;
ptrConfigPage^.aiRTrigActionPanelRight[5]:=10000 + gT_PageNumber.iHandMode_ConfigPosition;
ptrConfigPage^.aiFTrigActionPanelRight[1]:=0;
ptrConfigPage^.aiFTrigActionPanelRight[2]:=0;
ptrConfigPage^.aiFTrigActionPanelRight[3]:=0;
ptrConfigPage^.aiFTrigActionPanelRight[4]:=0;
ptrConfigPage^.aiFTrigActionPanelRight[5]:=0;
ptrConfigPage^.aiRTrigActionFunctionPanel[1]:=181;	(* Auswahl Position Führungsrohr *)
ptrConfigPage^.aiRTrigActionFunctionPanel[2]:=182;	(* Auswahl Abstand Führungsrohr *)
ptrConfigPage^.aiRTrigActionFunctionPanel[3]:=183;	(* Auswahl Werkzeug *)
ptrConfigPage^.aiRTrigActionFunctionPanel[4]:=184;	(* Auswahl Führungsrohr Einsatz *)
ptrConfigPage^.aiRTrigActionFunctionPanel[5]:=185;	(* KonfigPos EIN/AUS *)
ptrConfigPage^.aiRTrigActionFunctionPanel[6]:=186;	(* Speichern der Positionskonfiguration *)
ptrConfigPage^.aiRTrigActionFunctionPanel[7]:=0;
ptrConfigPage^.aiRTrigActionFunctionPanel[8]:=0;
ptrConfigPage^.aiRTrigActionFunctionPanel[9]:=0;
ptrConfigPage^.aiRTrigActionFunctionPanel[10]:=0;
ptrConfigPage^.aiRTrigActionFunctionPanel[11]:=0;
ptrConfigPage^.aiRTrigActionFunctionPanel[12]:=0;
TaskBar_SetupModeA;
ptrConfigPage^.xMaskBtStart:=TRUE;
ptrConfigPage^.xMaskBtStop:=TRUE;
END_ACTION
ACTION Page_120_HandMode_ProfileMngmt1:
(* QVis page 130, HandMode ProfileMngmt1 *)
iIndexPage:=gT_PageNumber.iHandMode_ProfileMngmt1;
iPageNumber:=iPageNumber+1;
T_Visu.T_PageIndex[iIndexPage].iIndexConfigPage:=iPageNumber;
ptrConfigPage:=ADR(T_Visu.T_ConfigPage[T_Visu.T_PageIndex[iIndexPage].iIndexConfigPage]);
ptrConfigPage^.sName:='HandMode ProfileMngmt1';
ptrConfigPage^.wMaskBtPanelLeft:=16#19;	(* SetupModeA, Parameter *)
ptrConfigPage^.wMaskBtPanelRight:=16#E0;	(* Profil laden, Profil speichern, Profil löschen, Page Up, Page Down *)
ptrConfigPage^.wMaskFunctionPanel:=16#0;
(* Process mask *)
ptrConfigPage^.wMaskProcBtPanelLeft:=16#9;	(* SetupModeA, Parameter *)
ptrConfigPage^.wMaskProcBtPanelRight:=16#0;	(* Page Up, Page Down *)
ptrConfigPage^.wMaskProcFunctionPanel:=16#0;
(* Button edge action *)
ptrConfigPage^.aiRTrigActionPanelLeft[1]:=0;
ptrConfigPage^.aiRTrigActionPanelLeft[2]:=0;
ptrConfigPage^.aiRTrigActionPanelLeft[3]:=0;
ptrConfigPage^.aiRTrigActionPanelLeft[4]:=0;
ptrConfigPage^.aiRTrigActionPanelLeft[5]:=11000 + gT_PageNumber.iHandMode_Parameter;		(* Parameter Page *)
ptrConfigPage^.aiRTrigActionPanelRight[1]:=1003;		(* Profil laden *)
ptrConfigPage^.aiRTrigActionPanelRight[2]:=1004;		(* Profil speichern *)
ptrConfigPage^.aiRTrigActionPanelRight[3]:=1005;		(* Profil löschen *)
ptrConfigPage^.aiRTrigActionPanelRight[4]:=0;
ptrConfigPage^.aiRTrigActionPanelRight[5]:=0;
ptrConfigPage^.aiFTrigActionPanelRight[1]:=0;
ptrConfigPage^.aiFTrigActionPanelRight[2]:=0;
ptrConfigPage^.aiFTrigActionPanelRight[3]:=0;
ptrConfigPage^.aiFTrigActionPanelRight[4]:=0;
ptrConfigPage^.aiFTrigActionPanelRight[5]:=0;
ptrConfigPage^.aiRTrigActionFunctionPanel[1]:=0;
ptrConfigPage^.aiRTrigActionFunctionPanel[2]:=0;
ptrConfigPage^.aiRTrigActionFunctionPanel[3]:=0;
ptrConfigPage^.aiRTrigActionFunctionPanel[4]:=0;
ptrConfigPage^.aiRTrigActionFunctionPanel[5]:=0;
ptrConfigPage^.aiRTrigActionFunctionPanel[6]:=0;
ptrConfigPage^.aiRTrigActionFunctionPanel[7]:=0;
ptrConfigPage^.aiRTrigActionFunctionPanel[8]:=0;
ptrConfigPage^.aiRTrigActionFunctionPanel[9]:=0;
ptrConfigPage^.aiRTrigActionFunctionPanel[10]:=0;
ptrConfigPage^.aiRTrigActionFunctionPanel[11]:=0;
ptrConfigPage^.aiRTrigActionFunctionPanel[12]:=0;
TaskBar_SetupModeA;
ptrConfigPage^.xMaskBtStart:=FALSE;
ptrConfigPage^.xMaskBtStop:=TRUE;
END_ACTION
ACTION Page_150_HandMode_Setup1:
(* QVis page 150, HandMode Setup1 *)
iIndexPage:=gT_PageNumber.iHandMode_Setup1;
iPageNumber:=iPageNumber+1;
T_Visu.T_PageIndex[iIndexPage].iIndexConfigPage:=iPageNumber;
ptrConfigPage:=ADR(T_Visu.T_ConfigPage[T_Visu.T_PageIndex[iIndexPage].iIndexConfigPage]);
ptrConfigPage^.sName:='HandMode Setup1';
ptrConfigPage^.wMaskBtPanelLeft:=16#19;	(* SetupModeA, Parameter *)
ptrConfigPage^.wMaskBtPanelRight:=16#0;
ptrConfigPage^.wMaskFunctionPanel:=16#0;	(* Einrichtung starten, Werte speichern *)
(* Process mask *)
ptrConfigPage^.wMaskProcBtPanelLeft:=16#9;	(* SetupModeA, Parameter *)
ptrConfigPage^.wMaskProcBtPanelRight:=16#0;
ptrConfigPage^.wMaskProcFunctionPanel:=16#0;
(* Button edge action *)
ptrConfigPage^.aiRTrigActionPanelLeft[1]:=0;
ptrConfigPage^.aiRTrigActionPanelLeft[2]:=0;
ptrConfigPage^.aiRTrigActionPanelLeft[3]:=0;
ptrConfigPage^.aiRTrigActionPanelLeft[4]:=0;
ptrConfigPage^.aiRTrigActionPanelLeft[5]:=11000 + gT_PageNumber.iHandMode_Parameter;		(* Parameter Page *)
ptrConfigPage^.aiRTrigActionPanelRight[1]:=0;
ptrConfigPage^.aiRTrigActionPanelRight[2]:=0;
ptrConfigPage^.aiRTrigActionPanelRight[3]:=0;
ptrConfigPage^.aiRTrigActionPanelRight[4]:=0;
ptrConfigPage^.aiRTrigActionPanelRight[5]:=0;
ptrConfigPage^.aiFTrigActionPanelRight[1]:=0;
ptrConfigPage^.aiFTrigActionPanelRight[2]:=0;
ptrConfigPage^.aiFTrigActionPanelRight[3]:=0;
ptrConfigPage^.aiFTrigActionPanelRight[4]:=0;
ptrConfigPage^.aiFTrigActionPanelRight[5]:=0;
ptrConfigPage^.aiRTrigActionFunctionPanel[1]:=170;(* Einrichtung Potentiometer starten *)
ptrConfigPage^.aiRTrigActionFunctionPanel[2]:=0;
ptrConfigPage^.aiRTrigActionFunctionPanel[3]:=0;
ptrConfigPage^.aiRTrigActionFunctionPanel[4]:=0;
ptrConfigPage^.aiRTrigActionFunctionPanel[5]:=0;
ptrConfigPage^.aiRTrigActionFunctionPanel[6]:=0;
ptrConfigPage^.aiRTrigActionFunctionPanel[7]:=0;
ptrConfigPage^.aiRTrigActionFunctionPanel[8]:=0;
ptrConfigPage^.aiRTrigActionFunctionPanel[9]:=0;
ptrConfigPage^.aiRTrigActionFunctionPanel[10]:=0;
ptrConfigPage^.aiRTrigActionFunctionPanel[11]:=0;
ptrConfigPage^.aiRTrigActionFunctionPanel[12]:=0;
TaskBar_SetupModeA;
ptrConfigPage^.xMaskBtStart:=TRUE;
ptrConfigPage^.xMaskBtStop:=TRUE;
END_ACTION
ACTION Page_160_HandMode_ErrorList:
(* QVis page 160, HandMode ErrorList *)
iIndexPage:=gT_PageNumber.iHandMode_ErrorList;
iPageNumber:=iPageNumber+1;
T_Visu.T_PageIndex[iIndexPage].iIndexConfigPage:=iPageNumber;
ptrConfigPage:=ADR(T_Visu.T_ConfigPage[T_Visu.T_PageIndex[iIndexPage].iIndexConfigPage]);
ptrConfigPage^.sName:='HandMode ErrorList';
ptrConfigPage^.wMaskBtPanelLeft:=16#19;	(* SetupModeA, Parameter *)
ptrConfigPage^.wMaskBtPanelRight:=16#60;	(* Reset Fehler, Löschen Fehlerliste *)
ptrConfigPage^.wMaskFunctionPanel:=16#0;
(* Process mask *)
ptrConfigPage^.wMaskProcBtPanelLeft:=16#9;	(* SetupModeA, Parameter *)
ptrConfigPage^.wMaskProcBtPanelRight:=16#0;
ptrConfigPage^.wMaskProcFunctionPanel:=16#0;
(* Button edge action *)
ptrConfigPage^.aiRTrigActionPanelLeft[1]:=0;
ptrConfigPage^.aiRTrigActionPanelLeft[2]:=0;
ptrConfigPage^.aiRTrigActionPanelLeft[3]:=0;
ptrConfigPage^.aiRTrigActionPanelLeft[4]:=0;
ptrConfigPage^.aiRTrigActionPanelLeft[5]:=11000 + gT_PageNumber.iHandMode_Parameter;		(* Parameter Page *)
ptrConfigPage^.aiRTrigActionPanelRight[1]:=99;		(* Reset Fehler *)
ptrConfigPage^.aiRTrigActionPanelRight[2]:=97;		(* Löschen Fehlerliste *)
ptrConfigPage^.aiRTrigActionPanelRight[3]:=0;
ptrConfigPage^.aiRTrigActionPanelRight[4]:=0;
ptrConfigPage^.aiRTrigActionPanelRight[5]:=0;
ptrConfigPage^.aiFTrigActionPanelRight[1]:=0;
ptrConfigPage^.aiFTrigActionPanelRight[2]:=0;
ptrConfigPage^.aiFTrigActionPanelRight[3]:=0;
ptrConfigPage^.aiFTrigActionPanelRight[4]:=0;
ptrConfigPage^.aiFTrigActionPanelRight[5]:=0;
ptrConfigPage^.aiRTrigActionFunctionPanel[1]:=0;
ptrConfigPage^.aiRTrigActionFunctionPanel[2]:=0;
ptrConfigPage^.aiRTrigActionFunctionPanel[3]:=0;
ptrConfigPage^.aiRTrigActionFunctionPanel[4]:=0;
ptrConfigPage^.aiRTrigActionFunctionPanel[5]:=0;
ptrConfigPage^.aiRTrigActionFunctionPanel[6]:=0;
ptrConfigPage^.aiRTrigActionFunctionPanel[7]:=0;
ptrConfigPage^.aiRTrigActionFunctionPanel[8]:=0;
ptrConfigPage^.aiRTrigActionFunctionPanel[9]:=0;
ptrConfigPage^.aiRTrigActionFunctionPanel[10]:=0;
ptrConfigPage^.aiRTrigActionFunctionPanel[11]:=0;
ptrConfigPage^.aiRTrigActionFunctionPanel[12]:=0;
TaskBar_SetupModeA;
ptrConfigPage^.xMaskBtStart:=FALSE;
ptrConfigPage^.xMaskBtStop:=TRUE;
END_ACTION
ACTION Page_170_HandMode_Parameter:
(* QVis page 170, HandMode Parameter *)
iIndexPage:=gT_PageNumber.iHandMode_Parameter;
iPageNumber:=iPageNumber+1;
T_Visu.T_PageIndex[iIndexPage].iIndexConfigPage:=iPageNumber;
ptrConfigPage:=ADR(T_Visu.T_ConfigPage[T_Visu.T_PageIndex[iIndexPage].iIndexConfigPage]);
ptrConfigPage^.sName:='HandMode Parameter';
ptrConfigPage^.wMaskBtPanelLeft:=16#19;	(* SetupModeA, Parameter *)
ptrConfigPage^.wMaskBtPanelRight:=16#200;	(* Speichern *)
ptrConfigPage^.wMaskFunctionPanel:=16#0;
(* Process mask *)
ptrConfigPage^.wMaskProcBtPanelLeft:=16#9;	(* SetupModeA, Parameter *)
ptrConfigPage^.wMaskProcBtPanelRight:=16#200;	(* Speichern *)
ptrConfigPage^.wMaskProcFunctionPanel:=16#0;
(* Button edge action *)
ptrConfigPage^.aiRTrigActionPanelLeft[1]:=0;
ptrConfigPage^.aiRTrigActionPanelLeft[2]:=0;
ptrConfigPage^.aiRTrigActionPanelLeft[3]:=0;
ptrConfigPage^.aiRTrigActionPanelLeft[4]:=0;
ptrConfigPage^.aiRTrigActionPanelLeft[5]:=5;		(* Parameter OFF-->Previous Page *)
ptrConfigPage^.aiRTrigActionPanelRight[1]:=0;
ptrConfigPage^.aiRTrigActionPanelRight[2]:=0;
ptrConfigPage^.aiRTrigActionPanelRight[3]:=0;
ptrConfigPage^.aiRTrigActionPanelRight[4]:=0;
ptrConfigPage^.aiRTrigActionPanelRight[5]:=1001;		(* Speichern *)
ptrConfigPage^.aiFTrigActionPanelRight[1]:=0;
ptrConfigPage^.aiFTrigActionPanelRight[2]:=0;
ptrConfigPage^.aiFTrigActionPanelRight[3]:=0;
ptrConfigPage^.aiFTrigActionPanelRight[4]:=0;
ptrConfigPage^.aiFTrigActionPanelRight[5]:=0;
ptrConfigPage^.aiRTrigActionFunctionPanel[1]:=0;
ptrConfigPage^.aiRTrigActionFunctionPanel[2]:=0;
ptrConfigPage^.aiRTrigActionFunctionPanel[3]:=0;
ptrConfigPage^.aiRTrigActionFunctionPanel[4]:=0;
ptrConfigPage^.aiRTrigActionFunctionPanel[5]:=0;
ptrConfigPage^.aiRTrigActionFunctionPanel[6]:=0;
ptrConfigPage^.aiRTrigActionFunctionPanel[7]:=0;
ptrConfigPage^.aiRTrigActionFunctionPanel[8]:=0;
ptrConfigPage^.aiRTrigActionFunctionPanel[9]:=0;
ptrConfigPage^.aiRTrigActionFunctionPanel[10]:=0;
ptrConfigPage^.aiRTrigActionFunctionPanel[11]:=0;
ptrConfigPage^.aiRTrigActionFunctionPanel[12]:=0;
TaskBar_SetupModeA;
ptrConfigPage^.xMaskBtStart:=FALSE;
ptrConfigPage^.xMaskBtStop:=TRUE;
END_ACTION
ACTION Page_210_WorkStation_Axis1:
(* QVis page 210, WorkStation Axis1 *)
iIndexPage:=gT_PageNumber.iWorkStation_Axis1;
iPageNumber:=iPageNumber+1;
T_Visu.T_PageIndex[iIndexPage].iIndexConfigPage:=iPageNumber;
ptrConfigPage:=ADR(T_Visu.T_ConfigPage[T_Visu.T_PageIndex[iIndexPage].iIndexConfigPage]);
ptrConfigPage^.sName:='WorkStation Axis1';
ptrConfigPage^.wMaskBtPanelLeft:=16#1A;	(* SetupModeB, Parameter *)
ptrConfigPage^.wMaskBtPanelRight:=16#0;	(* NegIncJogSlow, PosIncJogSlow, Page Up, Page Down *)
ptrConfigPage^.wMaskFunctionPanel:=16#3F;
(* Process mask *)
ptrConfigPage^.wMaskProcBtPanelLeft:=16#A;	(* SetupModeB, Parameter *)
ptrConfigPage^.wMaskProcBtPanelRight:=16#0;
ptrConfigPage^.wMaskProcFunctionPanel:=16#0;
(* Button edge action *)
ptrConfigPage^.aiRTrigActionPanelLeft[1]:=0;
ptrConfigPage^.aiRTrigActionPanelLeft[2]:=0;
ptrConfigPage^.aiRTrigActionPanelLeft[3]:=0;
ptrConfigPage^.aiRTrigActionPanelLeft[4]:=0;
ptrConfigPage^.aiRTrigActionPanelLeft[5]:=11000 + gT_PageNumber.iWorkStation_Parameter;		(* Parameter Page *)
ptrConfigPage^.aiRTrigActionPanelRight[1]:=217;		(* Achse Jog/Ink Bewegung -/- - *)
ptrConfigPage^.aiRTrigActionPanelRight[2]:=216;		(* Achse Jog/Ink Bewegung +/++ *)
ptrConfigPage^.aiRTrigActionPanelRight[3]:=0;
ptrConfigPage^.aiRTrigActionPanelRight[4]:=0;
ptrConfigPage^.aiRTrigActionPanelRight[5]:=0;
ptrConfigPage^.aiFTrigActionPanelRight[1]:=0;
ptrConfigPage^.aiFTrigActionPanelRight[2]:=0;
ptrConfigPage^.aiFTrigActionPanelRight[3]:=0;
ptrConfigPage^.aiFTrigActionPanelRight[4]:=0;
ptrConfigPage^.aiFTrigActionPanelRight[5]:=0;
ptrConfigPage^.aiRTrigActionFunctionPanel[1]:=203;
ptrConfigPage^.aiRTrigActionFunctionPanel[2]:=204;
ptrConfigPage^.aiRTrigActionFunctionPanel[3]:=0;
ptrConfigPage^.aiRTrigActionFunctionPanel[4]:=0;
ptrConfigPage^.aiRTrigActionFunctionPanel[5]:=185;	(* KonfigPos EIN/AUS *)
ptrConfigPage^.aiRTrigActionFunctionPanel[6]:=214;
ptrConfigPage^.aiRTrigActionFunctionPanel[7]:=0;
ptrConfigPage^.aiRTrigActionFunctionPanel[8]:=0;
ptrConfigPage^.aiRTrigActionFunctionPanel[9]:=0;
ptrConfigPage^.aiRTrigActionFunctionPanel[10]:=0;
ptrConfigPage^.aiRTrigActionFunctionPanel[11]:=0;
ptrConfigPage^.aiRTrigActionFunctionPanel[12]:=0;
TaskBar_SetupModeB;
ptrConfigPage^.xMaskBtStart:=TRUE;
ptrConfigPage^.xMaskBtStop:=TRUE;
END_ACTION
ACTION Page_220_WorkStation_Cylinder1:
(* QVis page 220, WorkStation Cylinder1 *)
iIndexPage:=gT_PageNumber.iWorkStation_Cylinder1;
iPageNumber:=iPageNumber+1;
T_Visu.T_PageIndex[iIndexPage].iIndexConfigPage:=iPageNumber;
ptrConfigPage:=ADR(T_Visu.T_ConfigPage[T_Visu.T_PageIndex[iIndexPage].iIndexConfigPage]);
ptrConfigPage^.sName:='WorkStation Cylinder1';
ptrConfigPage^.wMaskBtPanelLeft:=16#1A;	(* SetupModeB, Parameter *)
ptrConfigPage^.wMaskBtPanelRight:=16#60;	(* EIN,AUS, Drucklos *)
ptrConfigPage^.wMaskFunctionPanel:=16#0;
(* Process mask *)
ptrConfigPage^.wMaskProcBtPanelLeft:=16#A;	(* SetupModeB, Parameter *)
ptrConfigPage^.wMaskProcBtPanelRight:=16#0;
ptrConfigPage^.wMaskProcFunctionPanel:=16#0;
(* Button edge action *)
ptrConfigPage^.aiRTrigActionPanelLeft[1]:=0;
ptrConfigPage^.aiRTrigActionPanelLeft[2]:=0;
ptrConfigPage^.aiRTrigActionPanelLeft[3]:=0;
ptrConfigPage^.aiRTrigActionPanelLeft[4]:=0;
ptrConfigPage^.aiRTrigActionPanelLeft[5]:=11000 + gT_PageNumber.iWorkStation_Parameter;		(* Parameter Page *)
ptrConfigPage^.aiRTrigActionPanelRight[1]:=301;		(* EIN/AUS *)
ptrConfigPage^.aiRTrigActionPanelRight[2]:=302;		(* Zylinder Drucklos schalten *)
ptrConfigPage^.aiRTrigActionPanelRight[3]:=0;
ptrConfigPage^.aiRTrigActionPanelRight[4]:=0;
ptrConfigPage^.aiRTrigActionPanelRight[5]:=0;
ptrConfigPage^.aiFTrigActionPanelRight[1]:=0;
ptrConfigPage^.aiFTrigActionPanelRight[2]:=0;
ptrConfigPage^.aiFTrigActionPanelRight[3]:=0;
ptrConfigPage^.aiFTrigActionPanelRight[4]:=0;
ptrConfigPage^.aiFTrigActionPanelRight[5]:=0;
ptrConfigPage^.aiRTrigActionFunctionPanel[1]:=0;
ptrConfigPage^.aiRTrigActionFunctionPanel[2]:=0;
ptrConfigPage^.aiRTrigActionFunctionPanel[3]:=0;
ptrConfigPage^.aiRTrigActionFunctionPanel[4]:=0;
ptrConfigPage^.aiRTrigActionFunctionPanel[5]:=0;
ptrConfigPage^.aiRTrigActionFunctionPanel[6]:=0;
ptrConfigPage^.aiRTrigActionFunctionPanel[7]:=0;
ptrConfigPage^.aiRTrigActionFunctionPanel[8]:=0;
ptrConfigPage^.aiRTrigActionFunctionPanel[9]:=0;
ptrConfigPage^.aiRTrigActionFunctionPanel[10]:=0;
ptrConfigPage^.aiRTrigActionFunctionPanel[11]:=0;
ptrConfigPage^.aiRTrigActionFunctionPanel[12]:=0;
TaskBar_SetupModeB;
ptrConfigPage^.xMaskBtStart:=FALSE;
ptrConfigPage^.xMaskBtStop:=TRUE;
END_ACTION
ACTION Page_230_WorkStation_Valve1:
(* QVis page 230, WorkStation Valve1 *)
iIndexPage:=gT_PageNumber.iWorkStation_Valve1;
iPageNumber:=iPageNumber+1;
T_Visu.T_PageIndex[iIndexPage].iIndexConfigPage:=iPageNumber;
ptrConfigPage:=ADR(T_Visu.T_ConfigPage[T_Visu.T_PageIndex[iIndexPage].iIndexConfigPage]);
ptrConfigPage^.sName:='WorkStation Valve1';
ptrConfigPage^.wMaskBtPanelLeft:=16#1A;	(* SetupModeB, Parameter *)
ptrConfigPage^.wMaskBtPanelRight:=16#0;	(* wird dynamisch zugewiesen für EIN/AUS, wegen der Entgratstation *)
ptrConfigPage^.wMaskFunctionPanel:=16#0;
(* Process mask *)
ptrConfigPage^.wMaskProcBtPanelLeft:=16#A;	(* SetupModeB, Parameter *)
ptrConfigPage^.wMaskProcBtPanelRight:=16#0;
ptrConfigPage^.wMaskProcFunctionPanel:=16#0;
(* Button edge action *)
ptrConfigPage^.aiRTrigActionPanelLeft[1]:=0;
ptrConfigPage^.aiRTrigActionPanelLeft[2]:=0;
ptrConfigPage^.aiRTrigActionPanelLeft[3]:=0;
ptrConfigPage^.aiRTrigActionPanelLeft[4]:=0;
ptrConfigPage^.aiRTrigActionPanelLeft[5]:=11000 + gT_PageNumber.iWorkStation_Parameter;		(* Parameter Page *)
ptrConfigPage^.aiRTrigActionPanelRight[1]:=0;
ptrConfigPage^.aiRTrigActionPanelRight[2]:=0;
ptrConfigPage^.aiRTrigActionPanelRight[3]:=0;
ptrConfigPage^.aiRTrigActionPanelRight[4]:=0;
ptrConfigPage^.aiRTrigActionPanelRight[5]:=0;
ptrConfigPage^.aiFTrigActionPanelRight[1]:=0;
ptrConfigPage^.aiFTrigActionPanelRight[2]:=0;
ptrConfigPage^.aiFTrigActionPanelRight[3]:=0;
ptrConfigPage^.aiFTrigActionPanelRight[4]:=0;
ptrConfigPage^.aiFTrigActionPanelRight[5]:=0;
ptrConfigPage^.aiRTrigActionFunctionPanel[1]:=0;
ptrConfigPage^.aiRTrigActionFunctionPanel[2]:=0;
ptrConfigPage^.aiRTrigActionFunctionPanel[3]:=0;
ptrConfigPage^.aiRTrigActionFunctionPanel[4]:=0;
ptrConfigPage^.aiRTrigActionFunctionPanel[5]:=0;
ptrConfigPage^.aiRTrigActionFunctionPanel[6]:=0;
ptrConfigPage^.aiRTrigActionFunctionPanel[7]:=0;
ptrConfigPage^.aiRTrigActionFunctionPanel[8]:=0;
ptrConfigPage^.aiRTrigActionFunctionPanel[9]:=0;
ptrConfigPage^.aiRTrigActionFunctionPanel[10]:=0;
ptrConfigPage^.aiRTrigActionFunctionPanel[11]:=0;
ptrConfigPage^.aiRTrigActionFunctionPanel[12]:=0;
TaskBar_SetupModeB;
ptrConfigPage^.xMaskBtStart:=FALSE;
ptrConfigPage^.xMaskBtStop:=TRUE;
END_ACTION
ACTION Page_240_WorkStation_Function1:
(* QVis page 240, WorkStation Function1 *)
iIndexPage:=gT_PageNumber.iWorkStation_Function1;
iPageNumber:=iPageNumber+1;
T_Visu.T_PageIndex[iIndexPage].iIndexConfigPage:=iPageNumber;
ptrConfigPage:=ADR(T_Visu.T_ConfigPage[T_Visu.T_PageIndex[iIndexPage].iIndexConfigPage]);
ptrConfigPage^.sName:='WorkStation Function1';
ptrConfigPage^.wMaskBtPanelLeft:=16#1A;	(* SetupModeB, Parameter *)
ptrConfigPage^.wMaskBtPanelRight:=16#0;
ptrConfigPage^.wMaskFunctionPanel:=16#0;
(* Process mask *)
ptrConfigPage^.wMaskProcBtPanelLeft:=16#A;	(* SetupModeB, Parameter *)
ptrConfigPage^.wMaskProcBtPanelRight:=16#0;
ptrConfigPage^.wMaskProcFunctionPanel:=16#0;
(* Button edge action *)
ptrConfigPage^.aiRTrigActionPanelLeft[1]:=0;
ptrConfigPage^.aiRTrigActionPanelLeft[2]:=0;
ptrConfigPage^.aiRTrigActionPanelLeft[3]:=0;
ptrConfigPage^.aiRTrigActionPanelLeft[4]:=0;
ptrConfigPage^.aiRTrigActionPanelLeft[5]:=11000 + gT_PageNumber.iWorkStation_Parameter;		(* Parameter Page *)
ptrConfigPage^.aiRTrigActionPanelRight[1]:=0;
ptrConfigPage^.aiRTrigActionPanelRight[2]:=0;
ptrConfigPage^.aiRTrigActionPanelRight[3]:=0;
ptrConfigPage^.aiRTrigActionPanelRight[4]:=0;
ptrConfigPage^.aiRTrigActionPanelRight[5]:=0;
ptrConfigPage^.aiFTrigActionPanelRight[1]:=0;
ptrConfigPage^.aiFTrigActionPanelRight[2]:=0;
ptrConfigPage^.aiFTrigActionPanelRight[3]:=0;
ptrConfigPage^.aiFTrigActionPanelRight[4]:=0;
ptrConfigPage^.aiFTrigActionPanelRight[5]:=0;
ptrConfigPage^.aiRTrigActionFunctionPanel[1]:=0;
ptrConfigPage^.aiRTrigActionFunctionPanel[2]:=0;
ptrConfigPage^.aiRTrigActionFunctionPanel[3]:=0;
ptrConfigPage^.aiRTrigActionFunctionPanel[4]:=0;
ptrConfigPage^.aiRTrigActionFunctionPanel[5]:=0;
ptrConfigPage^.aiRTrigActionFunctionPanel[6]:=0;
ptrConfigPage^.aiRTrigActionFunctionPanel[7]:=0;
ptrConfigPage^.aiRTrigActionFunctionPanel[8]:=0;
ptrConfigPage^.aiRTrigActionFunctionPanel[9]:=0;
ptrConfigPage^.aiRTrigActionFunctionPanel[10]:=0;
ptrConfigPage^.aiRTrigActionFunctionPanel[11]:=0;
ptrConfigPage^.aiRTrigActionFunctionPanel[12]:=0;
TaskBar_SetupModeB;
ptrConfigPage^.xMaskBtStart:=TRUE;
ptrConfigPage^.xMaskBtStop:=TRUE;
END_ACTION
ACTION Page_250_WorkStation_Setup1:
(* QVis page 250, WorkStation Setup1 *)
iIndexPage:=gT_PageNumber.iWorkStation_Setup1;
iPageNumber:=iPageNumber+1;
T_Visu.T_PageIndex[iIndexPage].iIndexConfigPage:=iPageNumber;
ptrConfigPage:=ADR(T_Visu.T_ConfigPage[T_Visu.T_PageIndex[iIndexPage].iIndexConfigPage]);
ptrConfigPage^.sName:='WorkStation Setup1';
ptrConfigPage^.wMaskBtPanelLeft:=16#1A;	(* SetupModeB, Parameter *)
ptrConfigPage^.wMaskBtPanelRight:=16#3E0;
ptrConfigPage^.wMaskFunctionPanel:=16#0;
(* Process mask *)
ptrConfigPage^.wMaskProcBtPanelLeft:=16#A;	(* SetupModeB, Parameter *)
ptrConfigPage^.wMaskProcBtPanelRight:=16#3E0;
ptrConfigPage^.wMaskProcFunctionPanel:=16#0;
(* Button edge action *)
ptrConfigPage^.aiRTrigActionPanelLeft[1]:=0;
ptrConfigPage^.aiRTrigActionPanelLeft[2]:=0;
ptrConfigPage^.aiRTrigActionPanelLeft[3]:=0;
ptrConfigPage^.aiRTrigActionPanelLeft[4]:=0;
ptrConfigPage^.aiRTrigActionPanelLeft[5]:=11000 + gT_PageNumber.iWorkStation_Parameter;		(* Parameter Page *)
ptrConfigPage^.aiRTrigActionPanelRight[1]:=10000 + gT_PageNumber.iWorkStation_Setup1;
ptrConfigPage^.aiRTrigActionPanelRight[2]:=10000 + gT_PageNumber.iWorkStation_Setup2;
ptrConfigPage^.aiRTrigActionPanelRight[3]:=10000 + gT_PageNumber.iWorkStation_Setup3;
ptrConfigPage^.aiRTrigActionPanelRight[4]:=10000 + gT_PageNumber.iWorkStation_Setup4;
ptrConfigPage^.aiRTrigActionPanelRight[5]:=10000 + gT_PageNumber.iWorkStation_Setup5;
ptrConfigPage^.aiFTrigActionPanelRight[1]:=0;
ptrConfigPage^.aiFTrigActionPanelRight[2]:=0;
ptrConfigPage^.aiFTrigActionPanelRight[3]:=0;
ptrConfigPage^.aiFTrigActionPanelRight[4]:=0;
ptrConfigPage^.aiFTrigActionPanelRight[5]:=0;
ptrConfigPage^.aiRTrigActionFunctionPanel[1]:=0;
ptrConfigPage^.aiRTrigActionFunctionPanel[2]:=0;
ptrConfigPage^.aiRTrigActionFunctionPanel[3]:=0;
ptrConfigPage^.aiRTrigActionFunctionPanel[4]:=0;
ptrConfigPage^.aiRTrigActionFunctionPanel[5]:=0;
ptrConfigPage^.aiRTrigActionFunctionPanel[6]:=0;
ptrConfigPage^.aiRTrigActionFunctionPanel[7]:=0;
ptrConfigPage^.aiRTrigActionFunctionPanel[8]:=0;
ptrConfigPage^.aiRTrigActionFunctionPanel[9]:=0;
ptrConfigPage^.aiRTrigActionFunctionPanel[10]:=0;
ptrConfigPage^.aiRTrigActionFunctionPanel[11]:=0;
ptrConfigPage^.aiRTrigActionFunctionPanel[12]:=0;
TaskBar_SetupModeB;
ptrConfigPage^.xMaskBtStart:=TRUE;
ptrConfigPage^.xMaskBtStop:=TRUE;
END_ACTION
ACTION Page_251_WorkStation_Setup2:
(* QVis page 251, WorkStation Setup2 *)
iIndexPage:=gT_PageNumber.iWorkStation_Setup2;
iPageNumber:=iPageNumber+1;
T_Visu.T_PageIndex[iIndexPage].iIndexConfigPage:=iPageNumber;
ptrConfigPage:=ADR(T_Visu.T_ConfigPage[T_Visu.T_PageIndex[iIndexPage].iIndexConfigPage]);
ptrConfigPage^.sName:='WorkStation Setup2';
ptrConfigPage^.wMaskBtPanelLeft:=16#1A;	(* SetupModeB, Parameter *)
ptrConfigPage^.wMaskBtPanelRight:=16#3E0;
ptrConfigPage^.wMaskFunctionPanel:=16#0;
(* Process mask *)
ptrConfigPage^.wMaskProcBtPanelLeft:=16#A;	(* SetupModeB, Parameter *)
ptrConfigPage^.wMaskProcBtPanelRight:=16#3E0;
ptrConfigPage^.wMaskProcFunctionPanel:=16#0;
(* Button edge action *)
ptrConfigPage^.aiRTrigActionPanelLeft[1]:=0;
ptrConfigPage^.aiRTrigActionPanelLeft[2]:=0;
ptrConfigPage^.aiRTrigActionPanelLeft[3]:=0;
ptrConfigPage^.aiRTrigActionPanelLeft[4]:=0;
ptrConfigPage^.aiRTrigActionPanelLeft[5]:=11000 + gT_PageNumber.iWorkStation_Parameter;		(* Parameter Page *)
ptrConfigPage^.aiRTrigActionPanelRight[1]:=10000 + gT_PageNumber.iWorkStation_Setup1;
ptrConfigPage^.aiRTrigActionPanelRight[2]:=10000 + gT_PageNumber.iWorkStation_Setup2;
ptrConfigPage^.aiRTrigActionPanelRight[3]:=10000 + gT_PageNumber.iWorkStation_Setup3;
ptrConfigPage^.aiRTrigActionPanelRight[4]:=10000 + gT_PageNumber.iWorkStation_Setup4;
ptrConfigPage^.aiRTrigActionPanelRight[5]:=10000 + gT_PageNumber.iWorkStation_Setup5;
ptrConfigPage^.aiFTrigActionPanelRight[1]:=0;
ptrConfigPage^.aiFTrigActionPanelRight[2]:=0;
ptrConfigPage^.aiFTrigActionPanelRight[3]:=0;
ptrConfigPage^.aiFTrigActionPanelRight[4]:=0;
ptrConfigPage^.aiFTrigActionPanelRight[5]:=0;
ptrConfigPage^.aiRTrigActionFunctionPanel[1]:=0;
ptrConfigPage^.aiRTrigActionFunctionPanel[2]:=0;
ptrConfigPage^.aiRTrigActionFunctionPanel[3]:=0;
ptrConfigPage^.aiRTrigActionFunctionPanel[4]:=0;
ptrConfigPage^.aiRTrigActionFunctionPanel[5]:=0;
ptrConfigPage^.aiRTrigActionFunctionPanel[6]:=0;
ptrConfigPage^.aiRTrigActionFunctionPanel[7]:=0;
ptrConfigPage^.aiRTrigActionFunctionPanel[8]:=0;
ptrConfigPage^.aiRTrigActionFunctionPanel[9]:=0;
ptrConfigPage^.aiRTrigActionFunctionPanel[10]:=0;
ptrConfigPage^.aiRTrigActionFunctionPanel[11]:=0;
ptrConfigPage^.aiRTrigActionFunctionPanel[12]:=0;
TaskBar_SetupModeB;
ptrConfigPage^.xMaskBtStart:=TRUE;
ptrConfigPage^.xMaskBtStop:=TRUE;
END_ACTION
ACTION Page_252_WorkStation_Setup3:
(* QVis page 252, WorkStation Setup3 *)
iIndexPage:=gT_PageNumber.iWorkStation_Setup3;
iPageNumber:=iPageNumber+1;
T_Visu.T_PageIndex[iIndexPage].iIndexConfigPage:=iPageNumber;
ptrConfigPage:=ADR(T_Visu.T_ConfigPage[T_Visu.T_PageIndex[iIndexPage].iIndexConfigPage]);
ptrConfigPage^.sName:='WorkStation Setup3';
ptrConfigPage^.wMaskBtPanelLeft:=16#1A;	(* SetupModeB, Parameter *)
ptrConfigPage^.wMaskBtPanelRight:=16#3E0;
ptrConfigPage^.wMaskFunctionPanel:=16#0;
(* Process mask *)
ptrConfigPage^.wMaskProcBtPanelLeft:=16#A;	(* SetupModeB, Parameter *)
ptrConfigPage^.wMaskProcBtPanelRight:=16#3E0;
ptrConfigPage^.wMaskProcFunctionPanel:=16#0;
(* Button edge action *)
ptrConfigPage^.aiRTrigActionPanelLeft[1]:=0;
ptrConfigPage^.aiRTrigActionPanelLeft[2]:=0;
ptrConfigPage^.aiRTrigActionPanelLeft[3]:=0;
ptrConfigPage^.aiRTrigActionPanelLeft[4]:=0;
ptrConfigPage^.aiRTrigActionPanelLeft[5]:=11000 + gT_PageNumber.iWorkStation_Parameter;		(* Parameter Page *)
ptrConfigPage^.aiRTrigActionPanelRight[1]:=10000 + gT_PageNumber.iWorkStation_Setup1;
ptrConfigPage^.aiRTrigActionPanelRight[2]:=10000 + gT_PageNumber.iWorkStation_Setup2;
ptrConfigPage^.aiRTrigActionPanelRight[3]:=10000 + gT_PageNumber.iWorkStation_Setup3;
